LIN {X 0,Y 528.521,Z 608.402,A -85,B 0,C 180,E1 23622.926,E2 23622.926} C_VEL
LIN {X 0,Y 528.515,Z 608.398,A -85,B 0,C 180,E1 23619.468,E2 23619.468} C_VEL
LIN {X 0,Y 528.508,Z 608.399,A -85,B 0,C 180,E1 23616.041,E2 23616.041} C_VEL
LIN {X 0,Y 528.521,Z 608.403,A -85,B 0,C 180,E1 23612.627,E2 23612.627} C_VEL
LIN {X 0,Y 528.529,Z 608.395,A -85,B 0,C 180,E1 23609.214,E2 23609.214} C_VEL
LIN {X 0,Y 528.495,Z 608.401,A -85,B 0,C 180,E1 23605.77,E2 23605.77} C_VEL
LIN {X 0,Y 528.522,Z 608.404,A -85,B 0,C 180,E1 23602.317,E2 23602.317} C_VEL
LIN {X 0,Y 528.519,Z 608.398,A -85,B 0,C 180,E1 23598.875,E2 23598.875} C_VEL
LIN {X 0,Y 528.48,Z 608.403,A -85,B 0,C 180,E1 23595.472,E2 23595.472} C_VEL
LIN {X 0,Y 528.523,Z 608.403,A -85,B 0,C 180,E1 23592.122,E2 23592.122} C_VEL
LIN {X 0,Y 528.485,Z 608.404,A -85,B 0,C 180,E1 23588.815,E2 23588.815} C_VEL
LIN {X 0,Y 528.558,Z 608.653,A -85,B 0,C 180,E1 23586.299,E2 23586.299} C_VEL
LIN {X 0,Y 531.147,Z 620.669,A -85,B 0,C 180,E1 23584.859,E2 23584.859} C_VEL
LIN {X 0,Y 531.113,Z 646.994,A -85,B 0,C 180,E1 23581.942,E2 23581.942} C_VEL
LIN {X 0,Y 530.812,Z 675.191,A -85,B 0,C 180,E1 23578.705,E2 23578.705} C_VEL
LIN {X 0,Y 530.502,Z 697.757,A -85,B 0,C 180,E1 23576.089,E2 23576.089} C_VEL
LIN {X 0,Y 531.315,Z 704.19,A -85,B 0,C 180,E1 23575.96,E2 23575.96} C_VEL
LIN {X 0,Y 530.592,Z 836.819,A -85,B 0,C 180,E1 23574.081,E2 23574.081} C_VEL
LIN {X 0,Y 530.428,Z 853.085,A -85,B 0,C 180,E1 23573.642,E2 23573.642} C_VEL
LIN {X 0,Y 530.169,Z 868.62,A -85,B 0,C 180,E1 23573.013,E2 23573.013} C_VEL
LIN {X 0,Y 529.83,Z 883.45,A -85,B 0,C 180,E1 23572.191,E2 23572.191} C_VEL
LIN {X 0,Y 529.463,Z 897.184,A -85,B 0,C 180,E1 23571.201,E2 23571.201} C_VEL
LIN {X 0,Y 529.097,Z 909.864,A -85,B 0,C 180,E1 23570.043,E2 23570.043} C_VEL
LIN {X 0,Y 528.754,Z 921.003,A -85,B 0,C 180,E1 23568.768,E2 23568.768} C_VEL
LIN {X 0,Y 528.457,Z 931.118,A -85,B 0,C 180,E1 23567.322,E2 23567.322} C_VEL
LIN {X 0,Y 528.239,Z 939.83,A -85,B 0,C 180,E1 23565.726,E2 23565.726} C_VEL
LIN {X 0,Y 528.101,Z 946.573,A -85,B 0,C 180,E1 23564.114,E2 23564.114} C_VEL
LIN {X 0,Y 528.006,Z 952.107,A -85,B 0,C 180,E1 23562.272,E2 23562.272} C_VEL
LIN {X 0,Y 528.005,Z 952.163,A -85,B 0,C 180,E1 23562.25,E2 23562.25} C_VEL
LIN {X 0,Y 526.984,Z 954.183,A -85,B 0,C 180,E1 23561.442,E2 23561.442} C_VEL
LIN {X 0,Y 522.729,Z 957.032,A -85,B 0,C 180,E1 23560.019,E2 23560.019} C_VEL
LIN {X 0,Y 520.31,Z 958.175,A -85,B 0,C 180,E1 23558.953,E2 23558.953} C_VEL
LIN {X 0,Y 520.045,Z 958.343,A -85,B 0,C 180,E1 23558.525,E2 23558.525} C_VEL
LIN {X 0,Y 520.041,Z 957.958,A -85,B 0,C 180,E1 23556.667,E2 23556.667} C_VEL
LIN {X 0,Y 520.063,Z 955.8,A -85,B 0,C 180,E1 23554.856,E2 23554.856} C_VEL
LIN {X 0,Y 520.12,Z 951.746,A -85,B 0,C 180,E1 23553.02,E2 23553.02} C_VEL
LIN {X 0,Y 520.236,Z 945.996,A -85,B 0,C 180,E1 23551.283,E2 23551.283} C_VEL
LIN {X 0,Y 520.411,Z 938.536,A -85,B 0,C 180,E1 23549.617,E2 23549.617} C_VEL
LIN {X 0,Y 520.663,Z 929.608,A -85,B 0,C 180,E1 23548.082,E2 23548.082} C_VEL
LIN {X 0,Y 521.01,Z 918.657,A -85,B 0,C 180,E1 23546.596,E2 23546.596} C_VEL
LIN {X 0,Y 521.408,Z 906.398,A -85,B 0,C 180,E1 23545.282,E2 23545.282} C_VEL
LIN {X 0,Y 521.806,Z 893.101,A -85,B 0,C 180,E1 23544.149,E2 23544.149} C_VEL
LIN {X 0,Y 522.198,Z 878.496,A -85,B 0,C 180,E1 23543.179,E2 23543.179} C_VEL
LIN {X 0,Y 522.544,Z 863.741,A -85,B 0,C 180,E1 23542.434,E2 23542.434} C_VEL
LIN {X 0,Y 522.797,Z 847.6,A -85,B 0,C 180,E1 23541.853,E2 23541.853} C_VEL
LIN {X 0,Y 522.937,Z 831.072,A -85,B 0,C 180,E1 23541.478,E2 23541.478} C_VEL
LIN {X 0,Y 523.508,Z 702.169,A -85,B 0,C 180,E1 23539.641,E2 23539.641} C_VEL
LIN {X 0,Y 522.522,Z 696.556,A -85,B 0,C 180,E1 23539.485,E2 23539.485} C_VEL
LIN {X 0,Y 523.125,Z 666.461,A -85,B 0,C 180,E1 23535.915,E2 23535.915} C_VEL
LIN {X 0,Y 523.521,Z 639.644,A -85,B 0,C 180,E1 23532.766,E2 23532.766} C_VEL
LIN {X 0,Y 523.551,Z 621.942,A -85,B 0,C 180,E1 23530.696,E2 23530.696} C_VEL
LIN {X 0,Y 520.538,Z 609.538,A -85,B 0,C 180,E1 23529.053,E2 23529.053} C_VEL
LIN {X 0,Y 520.56,Z 609.378,A -85,B 0,C 180,E1 23525.998,E2 23525.998} C_VEL
LIN {X 0,Y 520.521,Z 609.389,A -85,B 0,C 180,E1 23522.668,E2 23522.668} C_VEL
LIN {X 0,Y 520.586,Z 609.388,A -85,B 0,C 180,E1 23519.311,E2 23519.311} C_VEL
LIN {X 0,Y 520.535,Z 609.391,A -85,B 0,C 180,E1 23515.979,E2 23515.979} C_VEL
LIN {X 0,Y 520.536,Z 609.392,A -85,B 0,C 180,E1 23512.473,E2 23512.473} C_VEL
LIN {X 0,Y 520.583,Z 609.379,A -85,B 0,C 180,E1 23509.174,E2 23509.174} C_VEL
LIN {X 0,Y 520.532,Z 609.381,A -85,B 0,C 180,E1 23505.829,E2 23505.829} C_VEL
LIN {X 0,Y 520.625,Z 609.66,A -85,B 0,C 180,E1 23502.669,E2 23502.669} C_VEL
LIN {X 0,Y 524.764,Z 625.278,A -85,B 0,C 180,E1 23500.318,E2 23500.318} C_VEL
LIN {X 0,Y 523.759,Z 651.946,A -85,B 0,C 180,E1 23496.908,E2 23496.908} C_VEL
LIN {X 0,Y 522.864,Z 678.978,A -85,B 0,C 180,E1 23493.509,E2 23493.509} C_VEL
LIN {X 0,Y 522.468,Z 693.224,A -85,B 0,C 180,E1 23491.755,E2 23491.755} C_VEL
LIN {X 0,Y 524.511,Z 704.529,A -85,B 0,C 180,E1 23491.475,E2 23491.475} C_VEL
LIN {X 0,Y 523.61,Z 835.562,A -85,B 0,C 180,E1 23489.587,E2 23489.587} C_VEL
LIN {X 0,Y 523.359,Z 852.526,A -85,B 0,C 180,E1 23489.121,E2 23489.121} C_VEL
LIN {X 0,Y 523.024,Z 867.254,A -85,B 0,C 180,E1 23488.521,E2 23488.521} C_VEL
LIN {X 0,Y 522.574,Z 882.116,A -85,B 0,C 180,E1 23487.698,E2 23487.698} C_VEL
LIN {X 0,Y 522.088,Z 896.006,A -85,B 0,C 180,E1 23486.707,E2 23486.707} C_VEL
LIN {X 0,Y 521.613,Z 908.793,A -85,B 0,C 180,E1 23485.548,E2 23485.548} C_VEL
LIN {X 0,Y 521.147,Z 920.994,A -85,B 0,C 180,E1 23484.164,E2 23484.164} C_VEL
LIN {X 0,Y 520.756,Z 931.108,A -85,B 0,C 180,E1 23482.72,E2 23482.72} C_VEL
LIN {X 0,Y 520.453,Z 940.34,A -85,B 0,C 180,E1 23481.048,E2 23481.048} C_VEL
LIN {X 0,Y 520.258,Z 947.386,A -85,B 0,C 180,E1 23479.368,E2 23479.368} C_VEL
LIN {X 0,Y 520.15,Z 952.932,A -85,B 0,C 180,E1 23477.557,E2 23477.557} C_VEL
LIN {X 0,Y 520.084,Z 956.511,A -85,B 0,C 180,E1 23475.755,E2 23475.755} C_VEL
LIN {X 0,Y 520.059,Z 958.338,A -85,B 0,C 180,E1 23473.928,E2 23473.928} C_VEL
LIN {X 0,Y 520.062,Z 958.416,A -85,B 0,C 180,E1 23472.085,E2 23472.085} C_VEL
LIN {X 0,Y 520.09,Z 956.657,A -85,B 0,C 180,E1 23470.224,E2 23470.224} C_VEL
LIN {X 0,Y 520.157,Z 953.294,A -85,B 0,C 180,E1 23468.461,E2 23468.461} C_VEL
LIN {X 0,Y 520.269,Z 947.993,A -85,B 0,C 180,E1 23466.679,E2 23466.679} C_VEL
LIN {X 0,Y 520.461,Z 941.165,A -85,B 0,C 180,E1 23464.999,E2 23464.999} C_VEL
LIN {X 0,Y 520.742,Z 932.761,A -85,B 0,C 180,E1 23463.425,E2 23463.425} C_VEL
LIN {X 0,Y 521.128,Z 922.872,A -85,B 0,C 180,E1 23461.955,E2 23461.955} C_VEL
LIN {X 0,Y 521.583,Z 911.544,A -85,B 0,C 180,E1 23460.611,E2 23460.611} C_VEL
LIN {X 0,Y 522.08,Z 898.49,A -85,B 0,C 180,E1 23459.374,E2 23459.374} C_VEL
LIN {X 0,Y 522.567,Z 885.129,A -85,B 0,C 180,E1 23458.37,E2 23458.37} C_VEL
LIN {X 0,Y 523.027,Z 870.3,A -85,B 0,C 180,E1 23457.508,E2 23457.508} C_VEL
LIN {X 0,Y 523.414,Z 855.24,A -85,B 0,C 180,E1 23456.852,E2 23456.852} C_VEL
LIN {X 0,Y 523.674,Z 839.22,A -85,B 0,C 180,E1 23456.375,E2 23456.375} C_VEL
LIN {X 0,Y 523.861,Z 816.787,A -85,B 0,C 180,E1 23455.998,E2 23455.998} C_VEL
LIN {X 0,Y 524.467,Z 702.284,A -85,B 0,C 180,E1 23454.351,E2 23454.351} C_VEL
LIN {X 0,Y 522.558,Z 693.202,A -85,B 0,C 180,E1 23454.094,E2 23454.094} C_VEL
LIN {X 0,Y 523.474,Z 665.562,A -85,B 0,C 180,E1 23450.644,E2 23450.644} C_VEL
LIN {X 0,Y 524.54,Z 637.445,A -85,B 0,C 180,E1 23447.052,E2 23447.052} C_VEL
LIN {X 0,Y 524.869,Z 625.09,A -85,B 0,C 180,E1 23445.436,E2 23445.436} C_VEL
LIN {X 0,Y 520.594,Z 609.506,A -85,B 0,C 180,E1 23442.986,E2 23442.986} C_VEL
LIN {X 0,Y 520.574,Z 609.387,A -85,B 0,C 180,E1 23439.456,E2 23439.456} C_VEL
LIN {X 0,Y 520.573,Z 609.389,A -85,B 0,C 180,E1 23435.997,E2 23435.997} C_VEL
LIN {X 0,Y 520.583,Z 609.393,A -85,B 0,C 180,E1 23432.524,E2 23432.524} C_VEL
LIN {X 0,Y 520.58,Z 609.385,A -85,B 0,C 180,E1 23429.074,E2 23429.074} C_VEL
LIN {X 0,Y 520.57,Z 609.385,A -85,B 0,C 180,E1 23425.605,E2 23425.605} C_VEL
LIN {X 0,Y 520.586,Z 609.386,A -85,B 0,C 180,E1 23422.114,E2 23422.114} C_VEL
LIN {X 0,Y 520.579,Z 609.382,A -85,B 0,C 180,E1 23418.593,E2 23418.593} C_VEL
LIN {X 0,Y 520.566,Z 609.383,A -85,B 0,C 180,E1 23415.143,E2 23415.143} C_VEL
LIN {X 0,Y 520.581,Z 609.391,A -85,B 0,C 180,E1 23411.635,E2 23411.635} C_VEL
LIN {X 0,Y 520.581,Z 609.385,A -85,B 0,C 180,E1 23408.171,E2 23408.171} C_VEL
LIN {X 0,Y 520.565,Z 609.386,A -85,B 0,C 180,E1 23404.738,E2 23404.738} C_VEL
LIN {X 0,Y 520.582,Z 609.385,A -85,B 0,C 180,E1 23401.321,E2 23401.321} C_VEL
LIN {X 0,Y 520.583,Z 609.384,A -85,B 0,C 180,E1 23397.799,E2 23397.799} C_VEL
LIN {X 0,Y 520.563,Z 609.387,A -85,B 0,C 180,E1 23394.379,E2 23394.379} C_VEL
LIN {X 0,Y 520.582,Z 609.382,A -85,B 0,C 180,E1 23390.939,E2 23390.939} C_VEL
LIN {X 0,Y 520.584,Z 609.383,A -85,B 0,C 180,E1 23387.465,E2 23387.465} C_VEL
LIN {X 0,Y 520.562,Z 609.391,A -85,B 0,C 180,E1 23384.058,E2 23384.058} C_VEL
LIN {X 0,Y 520.581,Z 609.38,A -85,B 0,C 180,E1 23380.71,E2 23380.71} C_VEL
LIN {X 0,Y 520.566,Z 609.381,A -85,B 0,C 180,E1 23377.29,E2 23377.29} C_VEL
LIN {X 0,Y 520.567,Z 609.387,A -85,B 0,C 180,E1 23373.762,E2 23373.762} C_VEL
LIN {X 0,Y 520.582,Z 609.389,A -85,B 0,C 180,E1 23370.296,E2 23370.296} C_VEL
LIN {X 0,Y 520.564,Z 609.387,A -85,B 0,C 180,E1 23366.87,E2 23366.87} C_VEL
LIN {X 0,Y 520.565,Z 609.391,A -85,B 0,C 180,E1 23363.32,E2 23363.32} C_VEL
LIN {X 0,Y 520.584,Z 609.389,A -85,B 0,C 180,E1 23359.953,E2 23359.953} C_VEL
LIN {X 0,Y 520.557,Z 609.385,A -85,B 0,C 180,E1 23356.555,E2 23356.555} C_VEL
LIN {X 0,Y 520.578,Z 609.392,A -85,B 0,C 180,E1 23353.126,E2 23353.126} C_VEL
LIN {X 0,Y 520.587,Z 609.386,A -85,B 0,C 180,E1 23349.63,E2 23349.63} C_VEL
LIN {X 0,Y 520.553,Z 609.393,A -85,B 0,C 180,E1 23346.223,E2 23346.223} C_VEL
LIN {X 0,Y 520.617,Z 609.623,A -85,B 0,C 180,E1 23345.548,E2 23345.548} C_VEL
LIN {X 0,Y 528.314,Z 631.638,A -85,B 0,C 180,E1 23343.125,E2 23343.125} C_VEL
LIN {X 0,Y 526.952,Z 675.578,A -85,B 0,C 180,E1 23339.685,E2 23339.685} C_VEL
LIN {X 0,Y 525.974,Z 709.847,A -85,B 0,C 180,E1 23337.075,E2 23337.075} C_VEL
LIN {X 0,Y 527.931,Z 723.514,A -85,B 0,C 180,E1 23336.758,E2 23336.758} C_VEL
LIN {X 0,Y 526.233,Z 927.53,A -85,B 0,C 180,E1 23333.802,E2 23333.802} C_VEL
LIN {X 0,Y 525.783,Z 946.957,A -85,B 0,C 180,E1 23333.314,E2 23333.314} C_VEL
LIN {X 0,Y 525.229,Z 964.796,A -85,B 0,C 180,E1 23332.674,E2 23332.674} C_VEL
LIN {X 0,Y 524.559,Z 982.787,A -85,B 0,C 180,E1 23331.82,E2 23331.82} C_VEL
LIN {X 0,Y 523.785,Z 1000.784,A -85,B 0,C 180,E1 23330.732,E2 23330.732} C_VEL
LIN {X 0,Y 523.028,Z 1017.39,A -85,B 0,C 180,E1 23329.492,E2 23329.492} C_VEL
LIN {X 0,Y 522.315,Z 1032.415,A -85,B 0,C 180,E1 23328.137,E2 23328.137} C_VEL
LIN {X 0,Y 521.648,Z 1046.702,A -85,B 0,C 180,E1 23326.592,E2 23326.592} C_VEL
LIN {X 0,Y 521.078,Z 1059.756,A -85,B 0,C 180,E1 23324.899,E2 23324.899} C_VEL
LIN {X 0,Y 520.633,Z 1071.3,A -85,B 0,C 180,E1 23323.098,E2 23323.098} C_VEL
LIN {X 0,Y 520.313,Z 1081.338,A -85,B 0,C 180,E1 23321.191,E2 23321.191} C_VEL
LIN {X 0,Y 520.102,Z 1089.433,A -85,B 0,C 180,E1 23319.293,E2 23319.293} C_VEL
LIN {X 0,Y 519.989,Z 1096.129,A -85,B 0,C 180,E1 23317.291,E2 23317.291} C_VEL
LIN {X 0,Y 519.926,Z 1101.295,A -85,B 0,C 180,E1 23315.185,E2 23315.185} C_VEL
LIN {X 0,Y 519.912,Z 1104.658,A -85,B 0,C 180,E1 23313.086,E2 23313.086} C_VEL
LIN {X 0,Y 519.908,Z 1106.304,A -85,B 0,C 180,E1 23310.991,E2 23310.991} C_VEL
LIN {X 0,Y 519.906,Z 1106.265,A -85,B 0,C 180,E1 23308.898,E2 23308.898} C_VEL
LIN {X 0,Y 519.914,Z 1104.539,A -85,B 0,C 180,E1 23306.803,E2 23306.803} C_VEL
LIN {X 0,Y 519.927,Z 1101.085,A -85,B 0,C 180,E1 23304.703,E2 23304.703} C_VEL
LIN {X 0,Y 519.992,Z 1095.818,A -85,B 0,C 180,E1 23302.598,E2 23302.598} C_VEL
LIN {X 0,Y 520.129,Z 1088.591,A -85,B 0,C 180,E1 23300.484,E2 23300.484} C_VEL
LIN {X 0,Y 520.358,Z 1079.733,A -85,B 0,C 180,E1 23298.472,E2 23298.472} C_VEL
LIN {X 0,Y 520.706,Z 1069.307,A -85,B 0,C 180,E1 23296.565,E2 23296.565} C_VEL
LIN {X 0,Y 521.168,Z 1057.586,A -85,B 0,C 180,E1 23294.797,E2 23294.797} C_VEL
LIN {X 0,Y 521.745,Z 1044.4,A -85,B 0,C 180,E1 23293.141,E2 23293.141} C_VEL
LIN {X 0,Y 522.396,Z 1030.569,A -85,B 0,C 180,E1 23291.684,E2 23291.684} C_VEL
LIN {X 0,Y 523.121,Z 1015.357,A -85,B 0,C 180,E1 23290.342,E2 23290.342} C_VEL
LIN {X 0,Y 523.869,Z 998.977,A -85,B 0,C 180,E1 23289.148,E2 23289.148} C_VEL
LIN {X 0,Y 524.599,Z 981.79,A -85,B 0,C 180,E1 23288.129,E2 23288.129} C_VEL
LIN {X 0,Y 525.255,Z 963.935,A -85,B 0,C 180,E1 23287.291,E2 23287.291} C_VEL
LIN {X 0,Y 525.829,Z 944.794,A -85,B 0,C 180,E1 23286.621,E2 23286.621} C_VEL
LIN {X 0,Y 526.261,Z 925.545,A -85,B 0,C 180,E1 23286.162,E2 23286.162} C_VEL
LIN {X 0,Y 527.774,Z 721.067,A -85,B 0,C 180,E1 23283.197,E2 23283.197} C_VEL
LIN {X 0,Y 525.911,Z 709.157,A -85,B 0,C 180,E1 23282.898,E2 23282.898} C_VEL
LIN {X 0,Y 527.325,Z 664.166,A -85,B 0,C 180,E1 23279.409,E2 23279.409} C_VEL
LIN {X 0,Y 528.418,Z 631.682,A -85,B 0,C 180,E1 23276.849,E2 23276.849} C_VEL
LIN {X 0,Y 520.631,Z 609.705,A -85,B 0,C 180,E1 23274.452,E2 23274.452} C_VEL
LIN {X 0,Y 520.581,Z 609.389,A -85,B 0,C 180,E1 23273.184,E2 23273.184} C_VEL
LIN {X 0,Y 520.563,Z 609.39,A -85,B 0,C 180,E1 23269.687,E2 23269.687} C_VEL
LIN {X 0,Y 520.582,Z 609.384,A -85,B 0,C 180,E1 23266.234,E2 23266.234} C_VEL
LIN {X 0,Y 520.58,Z 609.391,A -85,B 0,C 180,E1 23262.687,E2 23262.687} C_VEL
LIN {X 0,Y 520.573,Z 609.389,A -85,B 0,C 180,E1 23259.281,E2 23259.281} C_VEL
LIN {X 0,Y 520.574,Z 609.386,A -85,B 0,C 180,E1 23255.852,E2 23255.852} C_VEL
LIN {X 0,Y 520.569,Z 609.391,A -85,B 0,C 180,E1 23252.273,E2 23252.273} C_VEL
LIN {X 0,Y 520.583,Z 609.389,A -85,B 0,C 180,E1 23248.821,E2 23248.821} C_VEL
LIN {X 0,Y 520.571,Z 609.387,A -85,B 0,C 180,E1 23245.361,E2 23245.361} C_VEL
LIN {X 0,Y 520.556,Z 609.392,A -85,B 0,C 180,E1 23241.877,E2 23241.877} C_VEL
LIN {X 0,Y 520.588,Z 609.39,A -85,B 0,C 180,E1 23238.476,E2 23238.476} C_VEL
LIN {X 0,Y 520.547,Z 609.391,A -85,B 0,C 180,E1 23235.143,E2 23235.143} C_VEL
LIN {X 0,Y 520.546,Z 609.395,A -85,B 0,C 180,E1 23231.59,E2 23231.59} C_VEL
LIN {X 0,Y 520.59,Z 609.391,A -85,B 0,C 180,E1 23228.171,E2 23228.171} C_VEL
LIN {X 0,Y 520.576,Z 609.575,A -85,B 0,C 180,E1 23226.617,E2 23226.617} C_VEL
LIN {X 0,Y 523.556,Z 623.071,A -85,B 0,C 180,E1 23224.985,E2 23224.985} C_VEL
LIN {X 0,Y 523.519,Z 650.254,A -85,B 0,C 180,E1 23221.97,E2 23221.97} C_VEL
LIN {X 0,Y 523.179,Z 679.795,A -85,B 0,C 180,E1 23218.576,E2 23218.576} C_VEL
LIN {X 0,Y 522.952,Z 699.166,A -85,B 0,C 180,E1 23216.344,E2 23216.344} C_VEL
LIN {X 0,Y 523.715,Z 705.163,A -85,B 0,C 180,E1 23216.221,E2 23216.221} C_VEL
LIN {X 0,Y 522.897,Z 838.188,A -85,B 0,C 180,E1 23214.297,E2 23214.297} C_VEL
LIN {X 0,Y 522.743,Z 854.027,A -85,B 0,C 180,E1 23213.865,E2 23213.865} C_VEL
LIN {X 0,Y 522.484,Z 869.358,A -85,B 0,C 180,E1 23213.241,E2 23213.241} C_VEL
LIN {X 0,Y 522.159,Z 883.503,A -85,B 0,C 180,E1 23212.463,E2 23212.463} C_VEL
LIN {X 0,Y 521.753,Z 897.813,A -85,B 0,C 180,E1 23211.433,E2 23211.433} C_VEL
LIN {X 0,Y 521.369,Z 910.395,A -85,B 0,C 180,E1 23210.284,E2 23210.284} C_VEL
LIN {X 0,Y 520.977,Z 922.127,A -85,B 0,C 180,E1 23208.935,E2 23208.935} C_VEL
LIN {X 0,Y 520.646,Z 932.272,A -85,B 0,C 180,E1 23207.466,E2 23207.466} C_VEL
LIN {X 0,Y 520.402,Z 940.878,A -85,B 0,C 180,E1 23205.877,E2 23205.877} C_VEL
LIN {X 0,Y 520.243,Z 947.547,A -85,B 0,C 180,E1 23204.277,E2 23204.277} C_VEL
LIN {X 0,Y 520.123,Z 953.086,A -85,B 0,C 180,E1 23202.433,E2 23202.433} C_VEL
LIN {X 0,Y 520.066,Z 956.47,A -85,B 0,C 180,E1 23200.69,E2 23200.69} C_VEL
LIN {X 0,Y 520.042,Z 958.242,A -85,B 0,C 180,E1 23198.81,E2 23198.81} C_VEL
LIN {X 0,Y 520.045,Z 958.343,A -85,B 0,C 180,E1 23198.525,E2 23198.525} C_VEL
LIN {X 0,Y 519.064,Z 958.538,A -85,B 0,C 180,E1 23197.676,E2 23197.676} C_VEL
LIN {X 0,Y 514.653,Z 958.354,A -85,B 0,C 180,E1 23196.137,E2 23196.137} C_VEL
LIN {X 0,Y 512.417,Z 957.426,A -85,B 0,C 180,E1 23195.112,E2 23195.112} C_VEL
LIN {X 0,Y 512.16,Z 956.752,A -85,B 0,C 180,E1 23194.683,E2 23194.683} C_VEL
LIN {X 0,Y 512.236,Z 952.557,A -85,B 0,C 180,E1 23192.822,E2 23192.822} C_VEL
LIN {X 0,Y 512.369,Z 946.613,A -85,B 0,C 180,E1 23191.055,E2 23191.055} C_VEL
LIN {X 0,Y 512.573,Z 939.119,A -85,B 0,C 180,E1 23189.394,E2 23189.394} C_VEL
LIN {X 0,Y 512.867,Z 929.708,A -85,B 0,C 180,E1 23187.791,E2 23187.791} C_VEL
LIN {X 0,Y 513.246,Z 918.892,A -85,B 0,C 180,E1 23186.333,E2 23186.333} C_VEL
LIN {X 0,Y 513.67,Z 906.73,A -85,B 0,C 180,E1 23185.033,E2 23185.033} C_VEL
LIN {X 0,Y 514.072,Z 894.233,A -85,B 0,C 180,E1 23183.959,E2 23183.959} C_VEL
LIN {X 0,Y 514.47,Z 880.225,A -85,B 0,C 180,E1 23183.013,E2 23183.013} C_VEL
LIN {X 0,Y 514.849,Z 864.996,A -85,B 0,C 180,E1 23182.225,E2 23182.225} C_VEL
LIN {X 0,Y 515.107,Z 848.894,A -85,B 0,C 180,E1 23181.635,E2 23181.635} C_VEL
LIN {X 0,Y 515.252,Z 832.388,A -85,B 0,C 180,E1 23181.25,E2 23181.25} C_VEL
LIN {X 0,Y 515.9,Z 703.02,A -85,B 0,C 180,E1 23179.37,E2 23179.37} C_VEL
LIN {X 0,Y 514.903,Z 697.689,A -85,B 0,C 180,E1 23179.229,E2 23179.229} C_VEL
LIN {X 0,Y 515.501,Z 667.96,A -85,B 0,C 180,E1 23175.702,E2 23175.702} C_VEL
LIN {X 0,Y 515.964,Z 638.618,A -85,B 0,C 180,E1 23172.246,E2 23172.246} C_VEL
LIN {X 0,Y 515.968,Z 624.273,A -85,B 0,C 180,E1 23170.568,E2 23170.568} C_VEL
LIN {X 0,Y 512.598,Z 610.534,A -85,B 0,C 180,E1 23168.738,E2 23168.738} C_VEL
LIN {X 0,Y 512.635,Z 610.374,A -85,B 0,C 180,E1 23165.537,E2 23165.537} C_VEL
LIN {X 0,Y 512.595,Z 610.38,A -85,B 0,C 180,E1 23162.161,E2 23162.161} C_VEL
LIN {X 0,Y 512.591,Z 610.379,A -85,B 0,C 180,E1 23158.676,E2 23158.676} C_VEL
LIN {X 0,Y 512.641,Z 610.363,A -85,B 0,C 180,E1 23155.41,E2 23155.41} C_VEL
LIN {X 0,Y 512.591,Z 610.382,A -85,B 0,C 180,E1 23152.098,E2 23152.098} C_VEL
LIN {X 0,Y 512.626,Z 610.376,A -85,B 0,C 180,E1 23148.656,E2 23148.656} C_VEL
LIN {X 0,Y 512.626,Z 610.369,A -85,B 0,C 180,E1 23145.267,E2 23145.267} C_VEL
LIN {X 0,Y 512.676,Z 610.651,A -85,B 0,C 180,E1 23143.076,E2 23143.076} C_VEL
LIN {X 0,Y 517.224,Z 627.697,A -85,B 0,C 180,E1 23140.47,E2 23140.47} C_VEL
LIN {X 0,Y 516.176,Z 653.615,A -85,B 0,C 180,E1 23137.122,E2 23137.122} C_VEL
LIN {X 0,Y 515.201,Z 680.751,A -85,B 0,C 180,E1 23133.672,E2 23133.672} C_VEL
LIN {X 0,Y 514.831,Z 693.315,A -85,B 0,C 180,E1 23132.115,E2 23132.115} C_VEL
LIN {X 0,Y 517.116,Z 705.629,A -85,B 0,C 180,E1 23131.799,E2 23131.799} C_VEL
LIN {X 0,Y 516.122,Z 836.216,A -85,B 0,C 180,E1 23129.889,E2 23129.889} C_VEL
LIN {X 0,Y 515.853,Z 853.205,A -85,B 0,C 180,E1 23129.417,E2 23129.417} C_VEL
LIN {X 0,Y 515.472,Z 868.6,A -85,B 0,C 180,E1 23128.778,E2 23128.778} C_VEL
LIN {X 0,Y 514.985,Z 883.365,A -85,B 0,C 180,E1 23127.942,E2 23127.942} C_VEL
LIN {X 0,Y 514.456,Z 897.202,A -85,B 0,C 180,E1 23126.937,E2 23126.937} C_VEL
LIN {X 0,Y 513.93,Z 909.944,A -85,B 0,C 180,E1 23125.761,E2 23125.761} C_VEL
LIN {X 0,Y 513.414,Z 922.076,A -85,B 0,C 180,E1 23124.363,E2 23124.363} C_VEL
LIN {X 0,Y 512.99,Z 931.894,A -85,B 0,C 180,E1 23122.947,E2 23122.947} C_VEL
LIN {X 0,Y 512.634,Z 941.187,A -85,B 0,C 180,E1 23121.25,E2 23121.25} C_VEL
LIN {X 0,Y 512.4,Z 948.32,A -85,B 0,C 180,E1 23119.545,E2 23119.545} C_VEL
LIN {X 0,Y 512.266,Z 953.893,A -85,B 0,C 180,E1 23117.717,E2 23117.717} C_VEL
LIN {X 0,Y 512.187,Z 957.444,A -85,B 0,C 180,E1 23115.982,E2 23115.982} C_VEL
LIN {X 0,Y 512.15,Z 959.408,A -85,B 0,C 180,E1 23114.138,E2 23114.138} C_VEL
LIN {X 0,Y 512.15,Z 959.693,A -85,B 0,C 180,E1 23112.269,E2 23112.269} C_VEL
LIN {X 0,Y 512.183,Z 958.134,A -85,B 0,C 180,E1 23110.381,E2 23110.381} C_VEL
LIN {X 0,Y 512.267,Z 954.706,A -85,B 0,C 180,E1 23108.473,E2 23108.473} C_VEL
LIN {X 0,Y 512.394,Z 949.948,A -85,B 0,C 180,E1 23106.786,E2 23106.786} C_VEL
LIN {X 0,Y 512.62,Z 942.814,A -85,B 0,C 180,E1 23104.96,E2 23104.96} C_VEL
LIN {X 0,Y 512.944,Z 934.596,A -85,B 0,C 180,E1 23103.364,E2 23103.364} C_VEL
LIN {X 0,Y 513.406,Z 924.011,A -85,B 0,C 180,E1 23101.755,E2 23101.755} C_VEL
LIN {X 0,Y 513.916,Z 912.644,A -85,B 0,C 180,E1 23100.385,E2 23100.385} C_VEL
LIN {X 0,Y 514.467,Z 899.608,A -85,B 0,C 180,E1 23099.131,E2 23099.131} C_VEL
LIN {X 0,Y 514.997,Z 886.471,A -85,B 0,C 180,E1 23098.124,E2 23098.124} C_VEL
LIN {X 0,Y 515.503,Z 871.529,A -85,B 0,C 180,E1 23097.239,E2 23097.239} C_VEL
LIN {X 0,Y 515.941,Z 855.774,A -85,B 0,C 180,E1 23096.541,E2 23096.541} C_VEL
LIN {X 0,Y 516.213,Z 839.686,A -85,B 0,C 180,E1 23096.061,E2 23096.061} C_VEL
LIN {X 0,Y 516.413,Z 816.95,A -85,B 0,C 180,E1 23095.676,E2 23095.676} C_VEL
LIN {X 0,Y 517.106,Z 703.505,A -85,B 0,C 180,E1 23094.018,E2 23094.018} C_VEL
LIN {X 0,Y 514.98,Z 693.607,A -85,B 0,C 180,E1 23093.743,E2 23093.743} C_VEL
LIN {X 0,Y 515.872,Z 668.015,A -85,B 0,C 180,E1 23090.526,E2 23090.526} C_VEL
LIN {X 0,Y 517.05,Z 639.818,A -85,B 0,C 180,E1 23086.875,E2 23086.875} C_VEL
LIN {X 0,Y 517.462,Z 627.908,A -85,B 0,C 180,E1 23085.305,E2 23085.305} C_VEL
LIN {X 0,Y 512.672,Z 610.626,A -85,B 0,C 180,E1 23082.553,E2 23082.553} C_VEL
LIN {X 0,Y 512.632,Z 610.379,A -85,B 0,C 180,E1 23079.194,E2 23079.194} C_VEL
LIN {X 0,Y 512.643,Z 610.375,A -85,B 0,C 180,E1 23075.674,E2 23075.674} C_VEL
LIN {X 0,Y 512.637,Z 610.377,A -85,B 0,C 180,E1 23072.169,E2 23072.169} C_VEL
LIN {X 0,Y 512.636,Z 610.376,A -85,B 0,C 180,E1 23068.673,E2 23068.673} C_VEL
LIN {X 0,Y 512.643,Z 610.37,A -85,B 0,C 180,E1 23065.163,E2 23065.163} C_VEL
LIN {X 0,Y 512.634,Z 610.378,A -85,B 0,C 180,E1 23061.632,E2 23061.632} C_VEL
LIN {X 0,Y 512.637,Z 610.373,A -85,B 0,C 180,E1 23058.184,E2 23058.184} C_VEL
LIN {X 0,Y 512.649,Z 610.367,A -85,B 0,C 180,E1 23054.674,E2 23054.674} C_VEL
LIN {X 0,Y 512.628,Z 610.373,A -85,B 0,C 180,E1 23051.134,E2 23051.134} C_VEL
LIN {X 0,Y 512.643,Z 610.38,A -85,B 0,C 180,E1 23047.622,E2 23047.622} C_VEL
LIN {X 0,Y 512.642,Z 610.372,A -85,B 0,C 180,E1 23044.027,E2 23044.027} C_VEL
LIN {X 0,Y 512.625,Z 610.37,A -85,B 0,C 180,E1 23040.559,E2 23040.559} C_VEL
LIN {X 0,Y 512.643,Z 610.376,A -85,B 0,C 180,E1 23037.093,E2 23037.093} C_VEL
LIN {X 0,Y 512.644,Z 610.373,A -85,B 0,C 180,E1 23033.505,E2 23033.505} C_VEL
LIN {X 0,Y 512.624,Z 610.373,A -85,B 0,C 180,E1 23030.059,E2 23030.059} C_VEL
LIN {X 0,Y 512.644,Z 610.372,A -85,B 0,C 180,E1 23026.58,E2 23026.58} C_VEL
LIN {X 0,Y 512.645,Z 610.375,A -85,B 0,C 180,E1 23023.106,E2 23023.106} C_VEL
LIN {X 0,Y 512.623,Z 610.378,A -85,B 0,C 180,E1 23019.685,E2 23019.685} C_VEL
LIN {X 0,Y 512.643,Z 610.373,A -85,B 0,C 180,E1 23016.188,E2 23016.188} C_VEL
LIN {X 0,Y 512.645,Z 610.369,A -85,B 0,C 180,E1 23012.72,E2 23012.72} C_VEL
LIN {X 0,Y 512.619,Z 610.372,A -85,B 0,C 180,E1 23009.268,E2 23009.268} C_VEL
LIN {X 0,Y 512.646,Z 610.376,A -85,B 0,C 180,E1 23005.788,E2 23005.788} C_VEL
LIN {X 0,Y 512.647,Z 610.373,A -85,B 0,C 180,E1 23002.235,E2 23002.235} C_VEL
LIN {X 0,Y 512.617,Z 610.378,A -85,B 0,C 180,E1 22998.841,E2 22998.841} C_VEL
LIN {X 0,Y 512.645,Z 610.379,A -85,B 0,C 180,E1 22995.389,E2 22995.389} C_VEL
LIN {X 0,Y 512.644,Z 610.375,A -85,B 0,C 180,E1 22991.837,E2 22991.837} C_VEL
LIN {X 0,Y 512.614,Z 610.379,A -85,B 0,C 180,E1 22988.362,E2 22988.362} C_VEL
LIN {X 0,Y 512.657,Z 610.649,A -85,B 0,C 180,E1 22986.029,E2 22986.029} C_VEL
LIN {X 0,Y 519.677,Z 630.467,A -85,B 0,C 180,E1 22983.781,E2 22983.781} C_VEL
LIN {X 0,Y 521.03,Z 634.412,A -85,B 0,C 180,E1 22983.359,E2 22983.359} C_VEL
LIN {X 0,Y 519.493,Z 677.903,A -85,B 0,C 180,E1 22979.9,E2 22979.9} C_VEL
LIN {X 0,Y 518.492,Z 709.662,A -85,B 0,C 180,E1 22977.451,E2 22977.451} C_VEL
LIN {X 0,Y 520.724,Z 724.661,A -85,B 0,C 180,E1 22977.125,E2 22977.125} C_VEL
LIN {X 0,Y 518.917,Z 927.366,A -85,B 0,C 180,E1 22974.162,E2 22974.162} C_VEL
LIN {X 0,Y 518.422,Z 946.848,A -85,B 0,C 180,E1 22973.669,E2 22973.669} C_VEL
LIN {X 0,Y 517.796,Z 965.228,A -85,B 0,C 180,E1 22972.998,E2 22972.998} C_VEL
LIN {X 0,Y 517.076,Z 982.901,A -85,B 0,C 180,E1 22972.145,E2 22972.145} C_VEL
LIN {X 0,Y 516.233,Z 1000.7,A -85,B 0,C 180,E1 22971.056,E2 22971.056} C_VEL
LIN {X 0,Y 515.39,Z 1017.346,A -85,B 0,C 180,E1 22969.797,E2 22969.797} C_VEL
LIN {X 0,Y 514.59,Z 1032.543,A -85,B 0,C 180,E1 22968.405,E2 22968.405} C_VEL
LIN {X 0,Y 513.861,Z 1046.684,A -85,B 0,C 180,E1 22966.853,E2 22966.853} C_VEL
LIN {X 0,Y 513.225,Z 1059.757,A -85,B 0,C 180,E1 22965.133,E2 22965.133} C_VEL
LIN {X 0,Y 512.729,Z 1071.301,A -85,B 0,C 180,E1 22963.303,E2 22963.303} C_VEL
LIN {X 0,Y 512.364,Z 1081.339,A -85,B 0,C 180,E1 22961.367,E2 22961.367} C_VEL
LIN {X 0,Y 512.131,Z 1089.434,A -85,B 0,C 180,E1 22959.439,E2 22959.439} C_VEL
LIN {X 0,Y 511.997,Z 1096.129,A -85,B 0,C 180,E1 22957.405,E2 22957.405} C_VEL
LIN {X 0,Y 511.928,Z 1101.295,A -85,B 0,C 180,E1 22955.267,E2 22955.267} C_VEL
LIN {X 0,Y 511.913,Z 1104.657,A -85,B 0,C 180,E1 22953.135,E2 22953.135} C_VEL
LIN {X 0,Y 511.908,Z 1106.303,A -85,B 0,C 180,E1 22951.007,E2 22951.007} C_VEL
LIN {X 0,Y 511.906,Z 1106.265,A -85,B 0,C 180,E1 22948.881,E2 22948.881} C_VEL
LIN {X 0,Y 511.914,Z 1104.539,A -85,B 0,C 180,E1 22946.753,E2 22946.753} C_VEL
LIN {X 0,Y 511.931,Z 1101.085,A -85,B 0,C 180,E1 22944.62,E2 22944.62} C_VEL
LIN {X 0,Y 512.001,Z 1095.817,A -85,B 0,C 180,E1 22942.482,E2 22942.482} C_VEL
LIN {X 0,Y 512.159,Z 1088.59,A -85,B 0,C 180,E1 22940.334,E2 22940.334} C_VEL
LIN {X 0,Y 512.416,Z 1079.732,A -85,B 0,C 180,E1 22938.291,E2 22938.291} C_VEL
LIN {X 0,Y 512.806,Z 1069.306,A -85,B 0,C 180,E1 22936.354,E2 22936.354} C_VEL
LIN {X 0,Y 513.303,Z 1058.061,A -85,B 0,C 180,E1 22934.624,E2 22934.624} C_VEL
LIN {X 0,Y 513.952,Z 1044.739,A -85,B 0,C 180,E1 22932.916,E2 22932.916} C_VEL
LIN {X 0,Y 514.707,Z 1030.198,A -85,B 0,C 180,E1 22931.364,E2 22931.364} C_VEL
LIN {X 0,Y 515.515,Z 1014.819,A -85,B 0,C 180,E1 22929.996,E2 22929.996} C_VEL
LIN {X 0,Y 516.356,Z 998.084,A -85,B 0,C 180,E1 22928.77,E2 22928.77} C_VEL
LIN {X 0,Y 517.175,Z 980.554,A -85,B 0,C 180,E1 22927.732,E2 22927.732} C_VEL
LIN {X 0,Y 517.892,Z 962.601,A -85,B 0,C 180,E1 22926.896,E2 22926.896} C_VEL
LIN {X 0,Y 518.486,Z 944.051,A -85,B 0,C 180,E1 22926.248,E2 22926.248} C_VEL
LIN {X 0,Y 518.95,Z 924.903,A -85,B 0,C 180,E1 22925.793,E2 22925.793} C_VEL
LIN {X 0,Y 520.581,Z 722.325,A -85,B 0,C 180,E1 22922.834,E2 22922.834} C_VEL
LIN {X 0,Y 518.46,Z 708.947,A -85,B 0,C 180,E1 22922.513,E2 22922.513} C_VEL
LIN {X 0,Y 519.928,Z 664.783,A -85,B 0,C 180,E1 22919.058,E2 22919.058} C_VEL
LIN {X 0,Y 520.989,Z 634.108,A -85,B 0,C 180,E1 22916.598,E2 22916.598} C_VEL
LIN {X 0,Y 512.66,Z 610.644,A -85,B 0,C 180,E1 22913.951,E2 22913.951} C_VEL
LIN {X 0,Y 512.642,Z 610.381,A -85,B 0,C 180,E1 22910.742,E2 22910.742} C_VEL
LIN {X 0,Y 512.63,Z 610.379,A -85,B 0,C 180,E1 22907.334,E2 22907.334} C_VEL
LIN {X 0,Y 512.641,Z 610.372,A -85,B 0,C 180,E1 22903.809,E2 22903.809} C_VEL
LIN {X 0,Y 512.634,Z 610.378,A -85,B 0,C 180,E1 22900.304,E2 22900.304} C_VEL
LIN {X 0,Y 512.645,Z 610.381,A -85,B 0,C 180,E1 22896.782,E2 22896.782} C_VEL
LIN {X 0,Y 512.641,Z 610.376,A -85,B 0,C 180,E1 22893.203,E2 22893.203} C_VEL
LIN {X 0,Y 512.625,Z 610.376,A -85,B 0,C 180,E1 22889.777,E2 22889.777} C_VEL
LIN {X 0,Y 512.636,Z 610.381,A -85,B 0,C 180,E1 22886.279,E2 22886.279} C_VEL
LIN {X 0,Y 512.648,Z 610.376,A -85,B 0,C 180,E1 22882.838,E2 22882.838} C_VEL
LIN {X 0,Y 512.61,Z 610.379,A -85,B 0,C 180,E1 22879.484,E2 22879.484} C_VEL
LIN {X 0,Y 512.627,Z 610.383,A -85,B 0,C 180,E1 22875.963,E2 22875.963} C_VEL
LIN {X 0,Y 512.648,Z 610.379,A -85,B 0,C 180,E1 22872.503,E2 22872.503} C_VEL
LIN {X 0,Y 512.596,Z 610.384,A -85,B 0,C 180,E1 22869.09,E2 22869.09} C_VEL
LIN {X 0,Y 512.629,Z 610.629,A -85,B 0,C 180,E1 22866.915,E2 22866.915} C_VEL
LIN {X 0,Y 515.98,Z 624.52,A -85,B 0,C 180,E1 22865.225,E2 22865.225} C_VEL
LIN {X 0,Y 515.938,Z 651.595,A -85,B 0,C 180,E1 22862.221,E2 22862.221} C_VEL
LIN {X 0,Y 515.674,Z 678.805,A -85,B 0,C 180,E1 22859.111,E2 22859.111} C_VEL
LIN {X 0,Y 515.397,Z 700.47,A -85,B 0,C 180,E1 22856.611,E2 22856.611} C_VEL
LIN {X 0,Y 516.124,Z 706.055,A -85,B 0,C 180,E1 22856.491,E2 22856.491} C_VEL
LIN {X 0,Y 515.209,Z 839.561,A -85,B 0,C 180,E1 22854.519,E2 22854.519} C_VEL
LIN {X 0,Y 515.06,Z 855.37,A -85,B 0,C 180,E1 22854.08,E2 22854.08} C_VEL
LIN {X 0,Y 514.783,Z 871.287,A -85,B 0,C 180,E1 22853.419,E2 22853.419} C_VEL
LIN {X 0,Y 514.444,Z 885.26,A -85,B 0,C 180,E1 22852.63,E2 22852.63} C_VEL
LIN {X 0,Y 514.028,Z 899.164,A -85,B 0,C 180,E1 22851.611,E2 22851.611} C_VEL
LIN {X 0,Y 513.629,Z 911.459,A -85,B 0,C 180,E1 22850.475,E2 22850.475} C_VEL
LIN {X 0,Y 513.199,Z 923.318,A -85,B 0,C 180,E1 22849.095,E2 22849.095} C_VEL
LIN {X 0,Y 512.842,Z 933.351,A -85,B 0,C 180,E1 22847.629,E2 22847.629} C_VEL
LIN {X 0,Y 512.564,Z 942.062,A -85,B 0,C 180,E1 22846.002,E2 22846.002} C_VEL
LIN {X 0,Y 512.38,Z 948.748,A -85,B 0,C 180,E1 22844.378,E2 22844.378} C_VEL
LIN {X 0,Y 512.239,Z 954.301,A -85,B 0,C 180,E1 22842.506,E2 22842.506} C_VEL
LIN {X 0,Y 512.167,Z 957.687,A -85,B 0,C 180,E1 22840.736,E2 22840.736} C_VEL
LIN {X 0,Y 512.135,Z 959.453,A -85,B 0,C 180,E1 22838.827,E2 22838.827} C_VEL
LIN {X 0,Y 512.133,Z 959.374,A -85,B 0,C 180,E1 22837.016,E2 22837.016} C_VEL
LIN {X 0,Y 512.152,Z 957.383,A -85,B 0,C 180,E1 22835.058,E2 22835.058} C_VEL
LIN {X 0,Y 512.16,Z 956.752,A -85,B 0,C 180,E1 22834.683,E2 22834.683} C_VEL
LIN {X 0,Y 511.212,Z 955.242,A -85,B 0,C 180,E1 22833.838,E2 22833.838} C_VEL
LIN {X 0,Y 506.893,Z 952.009,A -85,B 0,C 180,E1 22832.316,E2 22832.316} C_VEL
LIN {X 0,Y 504.801,Z 949.294,A -85,B 0,C 180,E1 22831.381,E2 22831.381} C_VEL
LIN {X 0,Y 504.498,Z 947.579,A -85,B 0,C 180,E1 22830.914,E2 22830.914} C_VEL
LIN {X 0,Y 504.726,Z 940.198,A -85,B 0,C 180,E1 22829.263,E2 22829.263} C_VEL
LIN {X 0,Y 505.035,Z 931.071,A -85,B 0,C 180,E1 22827.687,E2 22827.687} C_VEL
LIN {X 0,Y 505.439,Z 920.492,A -85,B 0,C 180,E1 22826.229,E2 22826.229} C_VEL
LIN {X 0,Y 505.896,Z 908.224,A -85,B 0,C 180,E1 22824.891,E2 22824.891} C_VEL
LIN {X 0,Y 506.35,Z 895.07,A -85,B 0,C 180,E1 22823.743,E2 22823.743} C_VEL
LIN {X 0,Y 506.768,Z 881.221,A -85,B 0,C 180,E1 22822.797,E2 22822.797} C_VEL
LIN {X 0,Y 507.16,Z 866.176,A -85,B 0,C 180,E1 22822.007,E2 22822.007} C_VEL
LIN {X 0,Y 507.426,Z 850.025,A -85,B 0,C 180,E1 22821.406,E2 22821.406} C_VEL
LIN {X 0,Y 507.573,Z 833.555,A -85,B 0,C 180,E1 22821.014,E2 22821.014} C_VEL
LIN {X 0,Y 508.337,Z 704.093,A -85,B 0,C 180,E1 22819.095,E2 22819.095} C_VEL
LIN {X 0,Y 507.277,Z 698.44,A -85,B 0,C 180,E1 22818.932,E2 22818.932} C_VEL
LIN {X 0,Y 507.882,Z 669.181,A -85,B 0,C 180,E1 22815.453,E2 22815.453} C_VEL
LIN {X 0,Y 508.37,Z 640.299,A -85,B 0,C 180,E1 22812.036,E2 22812.036} C_VEL
LIN {X 0,Y 508.418,Z 626.698,A -85,B 0,C 180,E1 22810.44,E2 22810.44} C_VEL
LIN {X 0,Y 504.674,Z 611.527,A -85,B 0,C 180,E1 22808.411,E2 22808.411} C_VEL
LIN {X 0,Y 504.647,Z 611.373,A -85,B 0,C 180,E1 22804.889,E2 22804.889} C_VEL
LIN {X 0,Y 504.71,Z 611.369,A -85,B 0,C 180,E1 22801.534,E2 22801.534} C_VEL
LIN {X 0,Y 504.653,Z 611.369,A -85,B 0,C 180,E1 22798.155,E2 22798.155} C_VEL
LIN {X 0,Y 504.656,Z 611.35,A -85,B 0,C 180,E1 22794.576,E2 22794.576} C_VEL
LIN {X 0,Y 504.709,Z 611.362,A -85,B 0,C 180,E1 22791.256,E2 22791.256} C_VEL
LIN {X 0,Y 504.656,Z 611.372,A -85,B 0,C 180,E1 22787.885,E2 22787.885} C_VEL
LIN {X 0,Y 504.68,Z 611.373,A -85,B 0,C 180,E1 22784.35,E2 22784.35} C_VEL
LIN {X 0,Y 504.716,Z 611.708,A -85,B 0,C 180,E1 22783.487,E2 22783.487} C_VEL
LIN {X 0,Y 509.713,Z 630.183,A -85,B 0,C 180,E1 22780.626,E2 22780.626} C_VEL
LIN {X 0,Y 508.587,Z 656.234,A -85,B 0,C 180,E1 22777.228,E2 22777.228} C_VEL
LIN {X 0,Y 507.494,Z 683.369,A -85,B 0,C 180,E1 22773.728,E2 22773.728} C_VEL
LIN {X 0,Y 507.204,Z 693.359,A -85,B 0,C 180,E1 22772.486,E2 22772.486} C_VEL
LIN {X 0,Y 509.739,Z 706.736,A -85,B 0,C 180,E1 22772.133,E2 22772.133} C_VEL
LIN {X 0,Y 508.649,Z 837.036,A -85,B 0,C 180,E1 22770.197,E2 22770.197} C_VEL
LIN {X 0,Y 508.361,Z 853.994,A -85,B 0,C 180,E1 22769.719,E2 22769.719} C_VEL
LIN {X 0,Y 507.972,Z 868.85,A -85,B 0,C 180,E1 22769.098,E2 22769.098} C_VEL
LIN {X 0,Y 507.441,Z 883.757,A -85,B 0,C 180,E1 22768.25,E2 22768.25} C_VEL
LIN {X 0,Y 506.862,Z 897.7,A -85,B 0,C 180,E1 22767.23,E2 22767.23} C_VEL
LIN {X 0,Y 506.284,Z 910.565,A -85,B 0,C 180,E1 22766.037,E2 22766.037} C_VEL
LIN {X 0,Y 505.722,Z 922.376,A -85,B 0,C 180,E1 22764.668,E2 22764.668} C_VEL
LIN {X 0,Y 505.233,Z 932.682,A -85,B 0,C 180,E1 22763.181,E2 22763.181} C_VEL
LIN {X 0,Y 504.84,Z 941.477,A -85,B 0,C 180,E1 22761.573,E2 22761.573} C_VEL
LIN {X 0,Y 504.57,Z 948.847,A -85,B 0,C 180,E1 22759.842,E2 22759.842} C_VEL
LIN {X 0,Y 504.391,Z 954.584,A -85,B 0,C 180,E1 22757.987,E2 22757.987} C_VEL
LIN {X 0,Y 504.29,Z 958.49,A -85,B 0,C 180,E1 22756.119,E2 22756.119} C_VEL
LIN {X 0,Y 504.241,Z 960.549,A -85,B 0,C 180,E1 22754.237,E2 22754.237} C_VEL
LIN {X 0,Y 504.24,Z 960.9,A -85,B 0,C 180,E1 22752.339,E2 22752.339} C_VEL
LIN {X 0,Y 504.276,Z 959.609,A -85,B 0,C 180,E1 22750.543,E2 22750.543} C_VEL
LIN {X 0,Y 504.367,Z 956.364,A -85,B 0,C 180,E1 22748.607,E2 22748.607} C_VEL
LIN {X 0,Y 504.526,Z 951.486,A -85,B 0,C 180,E1 22746.773,E2 22746.773} C_VEL
LIN {X 0,Y 504.758,Z 944.997,A -85,B 0,C 180,E1 22745.044,E2 22745.044} C_VEL
LIN {X 0,Y 505.109,Z 937.105,A -85,B 0,C 180,E1 22743.426,E2 22743.426} C_VEL
LIN {X 0,Y 505.571,Z 927.594,A -85,B 0,C 180,E1 22741.891,E2 22741.891} C_VEL
LIN {X 0,Y 506.147,Z 916.014,A -85,B 0,C 180,E1 22740.406,E2 22740.406} C_VEL
LIN {X 0,Y 506.742,Z 903.612,A -85,B 0,C 180,E1 22739.136,E2 22739.136} C_VEL
LIN {X 0,Y 507.365,Z 889.407,A -85,B 0,C 180,E1 22737.987,E2 22737.987} C_VEL
LIN {X 0,Y 507.912,Z 875.219,A -85,B 0,C 180,E1 22737.09,E2 22737.09} C_VEL
LIN {X 0,Y 508.391,Z 859.533,A -85,B 0,C 180,E1 22736.35,E2 22736.35} C_VEL
LIN {X 0,Y 508.733,Z 843.265,A -85,B 0,C 180,E1 22735.81,E2 22735.81} C_VEL
LIN {X 0,Y 508.917,Z 825.252,A -85,B 0,C 180,E1 22735.464,E2 22735.464} C_VEL
LIN {X 0,Y 509.787,Z 704.872,A -85,B 0,C 180,E1 22733.675,E2 22733.675} C_VEL
LIN {X 0,Y 507.424,Z 693.852,A -85,B 0,C 180,E1 22733.362,E2 22733.362} C_VEL
LIN {X 0,Y 507.734,Z 683.565,A -85,B 0,C 180,E1 22732.091,E2 22732.091} C_VEL
LIN {X 0,Y 508.912,Z 656.244,A -85,B 0,C 180,E1 22728.54,E2 22728.54} C_VEL
LIN {X 0,Y 510.136,Z 630.971,A -85,B 0,C 180,E1 22725.196,E2 22725.196} C_VEL
LIN {X 0,Y 505.35,Z 613.717,A -85,B 0,C 180,E1 22722.43,E2 22722.43} C_VEL
LIN {X 0,Y 504.717,Z 611.456,A -85,B 0,C 180,E1 22721.992,E2 22721.992} C_VEL
LIN {X 0,Y 504.699,Z 611.367,A -85,B 0,C 180,E1 22718.468,E2 22718.468} C_VEL
LIN {X 0,Y 504.694,Z 611.368,A -85,B 0,C 180,E1 22715.067,E2 22715.067} C_VEL
LIN {X 0,Y 504.705,Z 611.359,A -85,B 0,C 180,E1 22711.534,E2 22711.534} C_VEL
LIN {X 0,Y 504.696,Z 611.369,A -85,B 0,C 180,E1 22707.924,E2 22707.924} C_VEL
LIN {X 0,Y 504.699,Z 611.364,A -85,B 0,C 180,E1 22704.46,E2 22704.46} C_VEL
LIN {X 0,Y 504.709,Z 611.362,A -85,B 0,C 180,E1 22700.891,E2 22700.891} C_VEL
LIN {X 0,Y 504.693,Z 611.368,A -85,B 0,C 180,E1 22697.407,E2 22697.407} C_VEL
LIN {X 0,Y 504.703,Z 611.36,A -85,B 0,C 180,E1 22693.87,E2 22693.87} C_VEL
LIN {X 0,Y 504.702,Z 611.358,A -85,B 0,C 180,E1 22690.271,E2 22690.271} C_VEL
LIN {X 0,Y 504.688,Z 611.363,A -85,B 0,C 180,E1 22686.827,E2 22686.827} C_VEL
LIN {X 0,Y 504.704,Z 611.37,A -85,B 0,C 180,E1 22683.294,E2 22683.294} C_VEL
LIN {X 0,Y 504.703,Z 611.357,A -85,B 0,C 180,E1 22679.773,E2 22679.773} C_VEL
LIN {X 0,Y 504.687,Z 611.355,A -85,B 0,C 180,E1 22676.252,E2 22676.252} C_VEL
LIN {X 0,Y 504.702,Z 611.365,A -85,B 0,C 180,E1 22672.716,E2 22672.716} C_VEL
LIN {X 0,Y 504.701,Z 611.362,A -85,B 0,C 180,E1 22669.152,E2 22669.152} C_VEL
LIN {X 0,Y 504.691,Z 611.357,A -85,B 0,C 180,E1 22665.643,E2 22665.643} C_VEL
LIN {X 0,Y 504.69,Z 611.36,A -85,B 0,C 180,E1 22662.117,E2 22662.117} C_VEL
LIN {X 0,Y 504.703,Z 611.367,A -85,B 0,C 180,E1 22658.608,E2 22658.608} C_VEL
LIN {X 0,Y 504.693,Z 611.364,A -85,B 0,C 180,E1 22655.142,E2 22655.142} C_VEL
LIN {X 0,Y 504.687,Z 611.369,A -85,B 0,C 180,E1 22651.597,E2 22651.597} C_VEL
LIN {X 0,Y 504.707,Z 611.359,A -85,B 0,C 180,E1 22648.198,E2 22648.198} C_VEL
LIN {X 0,Y 504.693,Z 611.361,A -85,B 0,C 180,E1 22644.656,E2 22644.656} C_VEL
LIN {X 0,Y 504.682,Z 611.37,A -85,B 0,C 180,E1 22641.095,E2 22641.095} C_VEL
LIN {X 0,Y 504.708,Z 611.368,A -85,B 0,C 180,E1 22637.641,E2 22637.641} C_VEL
LIN {X 0,Y 504.693,Z 611.364,A -85,B 0,C 180,E1 22634.179,E2 22634.179} C_VEL
LIN {X 0,Y 504.68,Z 611.37,A -85,B 0,C 180,E1 22630.643,E2 22630.643} C_VEL
LIN {X 0,Y 504.708,Z 611.369,A -85,B 0,C 180,E1 22627.173,E2 22627.173} C_VEL
LIN {X 0,Y 504.741,Z 611.78,A -85,B 0,C 180,E1 22626.505,E2 22626.505} C_VEL
LIN {X 0,Y 511.845,Z 631.853,A -85,B 0,C 180,E1 22624.18,E2 22624.18} C_VEL
LIN {X 0,Y 513.715,Z 637.665,A -85,B 0,C 180,E1 22623.556,E2 22623.556} C_VEL
LIN {X 0,Y 511.968,Z 680.767,A -85,B 0,C 180,E1 22620.062,E2 22620.062} C_VEL
LIN {X 0,Y 510.982,Z 709.594,A -85,B 0,C 180,E1 22617.809,E2 22617.809} C_VEL
LIN {X 0,Y 513.334,Z 725.798,A -85,B 0,C 180,E1 22617.452,E2 22617.452} C_VEL
LIN {X 0,Y 511.621,Z 927.16,A -85,B 0,C 180,E1 22614.533,E2 22614.533} C_VEL
LIN {X 0,Y 511.086,Z 946.631,A -85,B 0,C 180,E1 22614.038,E2 22614.038} C_VEL
LIN {X 0,Y 510.391,Z 965.395,A -85,B 0,C 180,E1 22613.343,E2 22613.343} C_VEL
LIN {X 0,Y 509.588,Z 983.364,A -85,B 0,C 180,E1 22612.46,E2 22612.46} C_VEL
LIN {X 0,Y 508.693,Z 1000.698,A -85,B 0,C 180,E1 22611.383,E2 22611.383} C_VEL
LIN {X 0,Y 507.801,Z 1016.785,A -85,B 0,C 180,E1 22610.156,E2 22610.156} C_VEL
LIN {X 0,Y 506.886,Z 1032.542,A -85,B 0,C 180,E1 22608.695,E2 22608.695} C_VEL
LIN {X 0,Y 506.08,Z 1046.684,A -85,B 0,C 180,E1 22607.12,E2 22607.12} C_VEL
LIN {X 0,Y 505.38,Z 1059.758,A -85,B 0,C 180,E1 22605.373,E2 22605.373} C_VEL
LIN {X 0,Y 504.816,Z 1071.553,A -85,B 0,C 180,E1 22603.47,E2 22603.47} C_VEL
LIN {X 0,Y 504.419,Z 1081.34,A -85,B 0,C 180,E1 22601.549,E2 22601.549} C_VEL
LIN {X 0,Y 504.164,Z 1089.434,A -85,B 0,C 180,E1 22599.589,E2 22599.589} C_VEL
LIN {X 0,Y 504.006,Z 1096.129,A -85,B 0,C 180,E1 22597.523,E2 22597.523} C_VEL
LIN {X 0,Y 503.932,Z 1101.294,A -85,B 0,C 180,E1 22595.351,E2 22595.351} C_VEL
LIN {X 0,Y 503.913,Z 1104.657,A -85,B 0,C 180,E1 22593.185,E2 22593.185} C_VEL
LIN {X 0,Y 503.908,Z 1106.303,A -85,B 0,C 180,E1 22591.023,E2 22591.023} C_VEL
LIN {X 0,Y 503.906,Z 1106.265,A -85,B 0,C 180,E1 22588.863,E2 22588.863} C_VEL
LIN {X 0,Y 503.914,Z 1104.539,A -85,B 0,C 180,E1 22586.701,E2 22586.701} C_VEL
LIN {X 0,Y 503.936,Z 1101.085,A -85,B 0,C 180,E1 22584.535,E2 22584.535} C_VEL
LIN {X 0,Y 504.012,Z 1095.817,A -85,B 0,C 180,E1 22582.362,E2 22582.362} C_VEL
LIN {X 0,Y 504.189,Z 1088.59,A -85,B 0,C 180,E1 22580.18,E2 22580.18} C_VEL
LIN {X 0,Y 504.48,Z 1079.732,A -85,B 0,C 180,E1 22578.104,E2 22578.104} C_VEL
LIN {X 0,Y 504.914,Z 1069.305,A -85,B 0,C 180,E1 22576.136,E2 22576.136} C_VEL
LIN {X 0,Y 505.46,Z 1058.165,A -85,B 0,C 180,E1 22574.393,E2 22574.393} C_VEL
LIN {X 0,Y 506.188,Z 1044.739,A -85,B 0,C 180,E1 22572.646,E2 22572.646} C_VEL
LIN {X 0,Y 507.019,Z 1030.196,A -85,B 0,C 180,E1 22571.07,E2 22571.07} C_VEL
LIN {X 0,Y 507.914,Z 1014.628,A -85,B 0,C 180,E1 22569.668,E2 22569.668} C_VEL
LIN {X 0,Y 508.826,Z 998.081,A -85,B 0,C 180,E1 22568.441,E2 22568.441} C_VEL
LIN {X 0,Y 509.721,Z 980.552,A -85,B 0,C 180,E1 22567.389,E2 22567.389} C_VEL
LIN {X 0,Y 510.508,Z 962.6,A -85,B 0,C 180,E1 22566.542,E2 22566.542} C_VEL
LIN {X 0,Y 511.15,Z 944.087,A -85,B 0,C 180,E1 22565.887,E2 22565.887} C_VEL
LIN {X 0,Y 511.647,Z 925.16,A -85,B 0,C 180,E1 22565.431,E2 22565.431} C_VEL
LIN {X 0,Y 513.195,Z 723.345,A -85,B 0,C 180,E1 22562.5,E2 22562.5} C_VEL
LIN {X 0,Y 510.966,Z 708.785,A -85,B 0,C 180,E1 22562.145,E2 22562.145} C_VEL
LIN {X 0,Y 512.54,Z 665.375,A -85,B 0,C 180,E1 22558.699,E2 22558.699} C_VEL
LIN {X 0,Y 513.71,Z 636.908,A -85,B 0,C 180,E1 22556.361,E2 22556.361} C_VEL
LIN {X 0,Y 505.141,Z 613.221,A -85,B 0,C 180,E1 22553.668,E2 22553.668} C_VEL
LIN {X 0,Y 504.716,Z 611.566,A -85,B 0,C 180,E1 22553.434,E2 22553.434} C_VEL
LIN {X 0,Y 504.693,Z 611.367,A -85,B 0,C 180,E1 22549.919,E2 22549.919} C_VEL
LIN {X 0,Y 504.702,Z 611.363,A -85,B 0,C 180,E1 22546.415,E2 22546.415} C_VEL
LIN {X 0,Y 504.705,Z 611.371,A -85,B 0,C 180,E1 22542.805,E2 22542.805} C_VEL
LIN {X 0,Y 504.697,Z 611.367,A -85,B 0,C 180,E1 22539.342,E2 22539.342} C_VEL
LIN {X 0,Y 504.696,Z 611.365,A -85,B 0,C 180,E1 22535.877,E2 22535.877} C_VEL
LIN {X 0,Y 504.695,Z 611.37,A -85,B 0,C 180,E1 22532.337,E2 22532.337} C_VEL
LIN {X 0,Y 504.706,Z 611.366,A -85,B 0,C 180,E1 22528.879,E2 22528.879} C_VEL
LIN {X 0,Y 504.695,Z 611.365,A -85,B 0,C 180,E1 22525.336,E2 22525.336} C_VEL
LIN {X 0,Y 504.679,Z 611.37,A -85,B 0,C 180,E1 22521.867,E2 22521.867} C_VEL
LIN {X 0,Y 504.709,Z 611.369,A -85,B 0,C 180,E1 22518.36,E2 22518.36} C_VEL
LIN {X 0,Y 504.682,Z 611.368,A -85,B 0,C 180,E1 22514.925,E2 22514.925} C_VEL
LIN {X 0,Y 504.662,Z 611.373,A -85,B 0,C 180,E1 22511.427,E2 22511.427} C_VEL
LIN {X 0,Y 504.708,Z 611.369,A -85,B 0,C 180,E1 22507.971,E2 22507.971} C_VEL
LIN {X 0,Y 504.7,Z 611.682,A -85,B 0,C 180,E1 22507.241,E2 22507.241} C_VEL
LIN {X 0,Y 508.399,Z 626.526,A -85,B 0,C 180,E1 22505.417,E2 22505.417} C_VEL
LIN {X 0,Y 508.404,Z 653.191,A -85,B 0,C 180,E1 22502.468,E2 22502.468} C_VEL
LIN {X 0,Y 508.101,Z 682.639,A -85,B 0,C 180,E1 22499.098,E2 22499.098} C_VEL
LIN {X 0,Y 507.872,Z 701.825,A -85,B 0,C 180,E1 22496.889,E2 22496.889} C_VEL
LIN {X 0,Y 508.557,Z 706.96,A -85,B 0,C 180,E1 22496.772,E2 22496.772} C_VEL
LIN {X 0,Y 507.528,Z 840.965,A -85,B 0,C 180,E1 22494.747,E2 22494.747} C_VEL
LIN {X 0,Y 507.384,Z 856.79,A -85,B 0,C 180,E1 22494.3,E2 22494.3} C_VEL
LIN {X 0,Y 507.113,Z 872.024,A -85,B 0,C 180,E1 22493.661,E2 22493.661} C_VEL
LIN {X 0,Y 506.763,Z 886.165,A -85,B 0,C 180,E1 22492.859,E2 22492.859} C_VEL
LIN {X 0,Y 506.321,Z 900.148,A -85,B 0,C 180,E1 22491.826,E2 22491.826} C_VEL
LIN {X 0,Y 505.895,Z 912.524,A -85,B 0,C 180,E1 22490.673,E2 22490.673} C_VEL
LIN {X 0,Y 505.431,Z 924.343,A -85,B 0,C 180,E1 22489.283,E2 22489.283} C_VEL
LIN {X 0,Y 505.065,Z 933.893,A -85,B 0,C 180,E1 22487.887,E2 22487.887} C_VEL
LIN {X 0,Y 504.742,Z 942.685,A -85,B 0,C 180,E1 22486.248,E2 22486.248} C_VEL
LIN {X 0,Y 504.534,Z 949.54,A -85,B 0,C 180,E1 22484.6,E2 22484.6} C_VEL
LIN {X 0,Y 504.366,Z 954.92,A -85,B 0,C 180,E1 22482.819,E2 22482.819} C_VEL
LIN {X 0,Y 504.279,Z 958.561,A -85,B 0,C 180,E1 22481.024,E2 22481.024} C_VEL
LIN {X 0,Y 504.236,Z 960.47,A -85,B 0,C 180,E1 22479.21,E2 22479.21} C_VEL
LIN {X 0,Y 504.222,Z 960.696,A -85,B 0,C 180,E1 22477.252,E2 22477.252} C_VEL
LIN {X 0,Y 504.238,Z 959.075,A -85,B 0,C 180,E1 22475.391,E2 22475.391} C_VEL
LIN {X 0,Y 504.299,Z 955.647,A -85,B 0,C 180,E1 22473.506,E2 22473.506} C_VEL
LIN {X 0,Y 504.417,Z 950.526,A -85,B 0,C 180,E1 22471.722,E2 22471.722} C_VEL
LIN {X 0,Y 504.498,Z 947.579,A -85,B 0,C 180,E1 22470.914,E2 22470.914} C_VEL
LIN {X 0,Y 503.61,Z 944.452,A -85,B 0,C 180,E1 22470.113,E2 22470.113} C_VEL
LIN {X 0,Y 499.135,Z 937.845,A -85,B 0,C 180,E1 22468.574,E2 22468.574} C_VEL
LIN {X 0,Y 497.367,Z 933.282,A -85,B 0,C 180,E1 22467.717,E2 22467.717} C_VEL
LIN {X 0,Y 497.253,Z 931.316,A -85,B 0,C 180,E1 22467.404,E2 22467.404} C_VEL
LIN {X 0,Y 497.681,Z 920.818,A -85,B 0,C 180,E1 22465.968,E2 22465.968} C_VEL
LIN {X 0,Y 498.199,Z 907.974,A -85,B 0,C 180,E1 22464.57,E2 22464.57} C_VEL
LIN {X 0,Y 498.663,Z 894.978,A -85,B 0,C 180,E1 22463.451,E2 22463.451} C_VEL
LIN {X 0,Y 499.14,Z 880.079,A -85,B 0,C 180,E1 22462.445,E2 22462.445} C_VEL
LIN {X 0,Y 499.52,Z 865.165,A -85,B 0,C 180,E1 22461.688,E2 22461.688} C_VEL
LIN {X 0,Y 499.8,Z 848.541,A -85,B 0,C 180,E1 22461.088,E2 22461.088} C_VEL
LIN {X 0,Y 499.914,Z 831.532,A -85,B 0,C 180,E1 22460.719,E2 22460.719} C_VEL
LIN {X 0,Y 500.767,Z 705.2,A -85,B 0,C 180,E1 22458.812,E2 22458.812} C_VEL
LIN {X 0,Y 499.676,Z 699.414,A -85,B 0,C 180,E1 22458.645,E2 22458.645} C_VEL
LIN {X 0,Y 500.304,Z 669.99,A -85,B 0,C 180,E1 22455.132,E2 22455.132} C_VEL
LIN {X 0,Y 500.79,Z 641.274,A -85,B 0,C 180,E1 22451.741,E2 22451.741} C_VEL
LIN {X 0,Y 500.759,Z 628.612,A -85,B 0,C 180,E1 22450.236,E2 22450.236} C_VEL
LIN {X 0,Y 496.764,Z 612.51,A -85,B 0,C 180,E1 22448.073,E2 22448.073} C_VEL
LIN {X 0,Y 496.705,Z 612.363,A -85,B 0,C 180,E1 22444.728,E2 22444.728} C_VEL
LIN {X 0,Y 496.752,Z 612.356,A -85,B 0,C 180,E1 22441.286,E2 22441.286} C_VEL
LIN {X 0,Y 496.727,Z 612.359,A -85,B 0,C 180,E1 22437.912,E2 22437.912} C_VEL
LIN {X 0,Y 496.711,Z 612.339,A -85,B 0,C 180,E1 22434.372,E2 22434.372} C_VEL
LIN {X 0,Y 496.765,Z 612.346,A -85,B 0,C 180,E1 22430.946,E2 22430.946} C_VEL
LIN {X 0,Y 496.738,Z 612.361,A -85,B 0,C 180,E1 22427.453,E2 22427.453} C_VEL
LIN {X 0,Y 496.739,Z 612.495,A -85,B 0,C 180,E1 22423.975,E2 22423.975} C_VEL
LIN {X 0,Y 501.637,Z 630.293,A -85,B 0,C 180,E1 22421.148,E2 22421.148} C_VEL
LIN {X 0,Y 502.186,Z 633.515,A -85,B 0,C 180,E1 22420.671,E2 22420.671} C_VEL
LIN {X 0,Y 500.938,Z 660.63,A -85,B 0,C 180,E1 22417.109,E2 22417.109} C_VEL
LIN {X 0,Y 499.697,Z 688.724,A -85,B 0,C 180,E1 22413.442,E2 22413.442} C_VEL
LIN {X 0,Y 499.621,Z 693.787,A -85,B 0,C 180,E1 22412.839,E2 22412.839} C_VEL
LIN {X 0,Y 502.365,Z 707.951,A -85,B 0,C 180,E1 22412.471,E2 22412.471} C_VEL
LIN {X 0,Y 501.187,Z 837.623,A -85,B 0,C 180,E1 22410.518,E2 22410.518} C_VEL
LIN {X 0,Y 500.883,Z 854.538,A -85,B 0,C 180,E1 22410.036,E2 22410.036} C_VEL
LIN {X 0,Y 500.443,Z 870.188,A -85,B 0,C 180,E1 22409.371,E2 22409.371} C_VEL
LIN {X 0,Y 499.875,Z 885.008,A -85,B 0,C 180,E1 22408.51,E2 22408.51} C_VEL
LIN {X 0,Y 499.252,Z 898.905,A -85,B 0,C 180,E1 22407.475,E2 22407.475} C_VEL
LIN {X 0,Y 498.619,Z 911.724,A -85,B 0,C 180,E1 22406.264,E2 22406.264} C_VEL
LIN {X 0,Y 497.979,Z 924.066,A -85,B 0,C 180,E1 22404.804,E2 22404.804} C_VEL
LIN {X 0,Y 497.444,Z 934.153,A -85,B 0,C 180,E1 22403.306,E2 22403.306} C_VEL
LIN {X 0,Y 496.992,Z 943.447,A -85,B 0,C 180,E1 22401.555,E2 22401.555} C_VEL
LIN {X 0,Y 496.687,Z 950.585,A -85,B 0,C 180,E1 22399.797,E2 22399.797} C_VEL
LIN {X 0,Y 496.497,Z 956.173,A -85,B 0,C 180,E1 22397.911,E2 22397.911} C_VEL
LIN {X 0,Y 496.378,Z 959.903,A -85,B 0,C 180,E1 22396.012,E2 22396.012} C_VEL
LIN {X 0,Y 496.329,Z 961.898,A -85,B 0,C 180,E1 22393.979,E2 22393.979} C_VEL
LIN {X 0,Y 496.333,Z 962.003,A -85,B 0,C 180,E1 22392.048,E2 22392.048} C_VEL
LIN {X 0,Y 496.386,Z 960.285,A -85,B 0,C 180,E1 22390.098,E2 22390.098} C_VEL
LIN {X 0,Y 496.513,Z 956.823,A -85,B 0,C 180,E1 22388.179,E2 22388.179} C_VEL
LIN {X 0,Y 496.712,Z 951.356,A -85,B 0,C 180,E1 22386.26,E2 22386.26} C_VEL
LIN {X 0,Y 497.026,Z 944.498,A -85,B 0,C 180,E1 22384.501,E2 22384.501} C_VEL
LIN {X 0,Y 497.445,Z 936.065,A -85,B 0,C 180,E1 22382.854,E2 22382.854} C_VEL
LIN {X 0,Y 498.021,Z 925.773,A -85,B 0,C 180,E1 22381.26,E2 22381.26} C_VEL
LIN {X 0,Y 498.643,Z 914.224,A -85,B 0,C 180,E1 22379.842,E2 22379.842} C_VEL
LIN {X 0,Y 499.329,Z 901.004,A -85,B 0,C 180,E1 22378.543,E2 22378.543} C_VEL
LIN {X 0,Y 499.946,Z 887.899,A -85,B 0,C 180,E1 22377.522,E2 22377.522} C_VEL
LIN {X 0,Y 500.545,Z 872.899,A -85,B 0,C 180,E1 22376.614,E2 22376.614} C_VEL
LIN {X 0,Y 501.039,Z 857.4,A -85,B 0,C 180,E1 22375.911,E2 22375.911} C_VEL
LIN {X 0,Y 501.352,Z 840.989,A -85,B 0,C 180,E1 22375.409,E2 22375.409} C_VEL
LIN {X 0,Y 501.588,Z 817.581,A -85,B 0,C 180,E1 22375.002,E2 22375.002} C_VEL
LIN {X 0,Y 502.492,Z 706.174,A -85,B 0,C 180,E1 22373.318,E2 22373.318} C_VEL
LIN {X 0,Y 499.858,Z 693.792,A -85,B 0,C 180,E1 22372.951,E2 22372.951} C_VEL
LIN {X 0,Y 500.993,Z 666.474,A -85,B 0,C 180,E1 22369.412,E2 22369.412} C_VEL
LIN {X 0,Y 502.398,Z 639.741,A -85,B 0,C 180,E1 22365.849,E2 22365.849} C_VEL
LIN {X 0,Y 502.554,Z 633.06,A -85,B 0,C 180,E1 22364.935,E2 22364.935} C_VEL
LIN {X 0,Y 498.275,Z 617.526,A -85,B 0,C 180,E1 22362.395,E2 22362.395} C_VEL
LIN {X 0,Y 496.766,Z 612.438,A -85,B 0,C 180,E1 22361.468,E2 22361.468} C_VEL
LIN {X 0,Y 496.758,Z 612.354,A -85,B 0,C 180,E1 22358.018,E2 22358.018} C_VEL
LIN {X 0,Y 496.762,Z 612.355,A -85,B 0,C 180,E1 22354.389,E2 22354.389} C_VEL
LIN {X 0,Y 496.755,Z 612.351,A -85,B 0,C 180,E1 22350.881,E2 22350.881} C_VEL
LIN {X 0,Y 496.765,Z 612.353,A -85,B 0,C 180,E1 22347.317,E2 22347.317} C_VEL
LIN {X 0,Y 496.755,Z 612.356,A -85,B 0,C 180,E1 22343.679,E2 22343.679} C_VEL
LIN {X 0,Y 496.765,Z 612.358,A -85,B 0,C 180,E1 22340.132,E2 22340.132} C_VEL
LIN {X 0,Y 496.763,Z 612.353,A -85,B 0,C 180,E1 22336.487,E2 22336.487} C_VEL
LIN {X 0,Y 496.752,Z 612.355,A -85,B 0,C 180,E1 22333.029,E2 22333.029} C_VEL
LIN {X 0,Y 496.764,Z 612.349,A -85,B 0,C 180,E1 22329.5,E2 22329.5} C_VEL
LIN {X 0,Y 496.763,Z 612.349,A -85,B 0,C 180,E1 22326.008,E2 22326.008} C_VEL
LIN {X 0,Y 496.754,Z 612.352,A -85,B 0,C 180,E1 22322.423,E2 22322.423} C_VEL
LIN {X 0,Y 496.758,Z 612.358,A -85,B 0,C 180,E1 22318.847,E2 22318.847} C_VEL
LIN {X 0,Y 496.761,Z 612.344,A -85,B 0,C 180,E1 22315.267,E2 22315.267} C_VEL
LIN {X 0,Y 496.767,Z 612.346,A -85,B 0,C 180,E1 22311.668,E2 22311.668} C_VEL
LIN {X 0,Y 496.747,Z 612.355,A -85,B 0,C 180,E1 22308.153,E2 22308.153} C_VEL
LIN {X 0,Y 496.768,Z 612.352,A -85,B 0,C 180,E1 22304.593,E2 22304.593} C_VEL
LIN {X 0,Y 496.766,Z 612.342,A -85,B 0,C 180,E1 22300.97,E2 22300.97} C_VEL
LIN {X 0,Y 496.744,Z 612.348,A -85,B 0,C 180,E1 22297.5,E2 22297.5} C_VEL
LIN {X 0,Y 496.761,Z 612.355,A -85,B 0,C 180,E1 22293.974,E2 22293.974} C_VEL
LIN {X 0,Y 496.768,Z 612.355,A -85,B 0,C 180,E1 22290.4,E2 22290.4} C_VEL
LIN {X 0,Y 496.75,Z 612.355,A -85,B 0,C 180,E1 22286.858,E2 22286.858} C_VEL
LIN {X 0,Y 496.746,Z 612.357,A -85,B 0,C 180,E1 22283.235,E2 22283.235} C_VEL
LIN {X 0,Y 496.769,Z 612.356,A -85,B 0,C 180,E1 22279.713,E2 22279.713} C_VEL
LIN {X 0,Y 496.765,Z 612.349,A -85,B 0,C 180,E1 22276.101,E2 22276.101} C_VEL
LIN {X 0,Y 496.738,Z 612.358,A -85,B 0,C 180,E1 22272.549,E2 22272.549} C_VEL
LIN {X 0,Y 496.77,Z 612.358,A -85,B 0,C 180,E1 22269.048,E2 22269.048} C_VEL
LIN {X 0,Y 496.806,Z 612.627,A -85,B 0,C 180,E1 22267.068,E2 22267.068} C_VEL
LIN {X 0,Y 503.23,Z 630.879,A -85,B 0,C 180,E1 22264.857,E2 22264.857} C_VEL
LIN {X 0,Y 506.422,Z 639.933,A -85,B 0,C 180,E1 22263.832,E2 22263.832} C_VEL
LIN {X 0,Y 504.394,Z 684.367,A -85,B 0,C 180,E1 22260.166,E2 22260.166} C_VEL
LIN {X 0,Y 503.463,Z 709.124,A -85,B 0,C 180,E1 22258.192,E2 22258.192} C_VEL
LIN {X 0,Y 505.962,Z 726.984,A -85,B 0,C 180,E1 22257.789,E2 22257.789} C_VEL
LIN {X 0,Y 504.114,Z 926.829,A -85,B 0,C 180,E1 22254.852,E2 22254.852} C_VEL
LIN {X 0,Y 503.556,Z 946.575,A -85,B 0,C 180,E1 22254.35,E2 22254.35} C_VEL
LIN {X 0,Y 502.854,Z 965.6,A -85,B 0,C 180,E1 22253.65,E2 22253.65} C_VEL
LIN {X 0,Y 502.056,Z 983.725,A -85,B 0,C 180,E1 22252.768,E2 22252.768} C_VEL
LIN {X 0,Y 501.22,Z 999.86,A -85,B 0,C 180,E1 22251.78,E2 22251.78} C_VEL
LIN {X 0,Y 500.195,Z 1016.783,A -85,B 0,C 180,E1 22250.476,E2 22250.476} C_VEL
LIN {X 0,Y 499.224,Z 1032.179,A -85,B 0,C 180,E1 22249.033,E2 22249.033} C_VEL
LIN {X 0,Y 498.311,Z 1046.684,A -85,B 0,C 180,E1 22247.395,E2 22247.395} C_VEL
LIN {X 0,Y 497.542,Z 1059.758,A -85,B 0,C 180,E1 22245.622,E2 22245.622} C_VEL
LIN {X 0,Y 496.929,Z 1071.302,A -85,B 0,C 180,E1 22243.734,E2 22243.734} C_VEL
LIN {X 0,Y 496.478,Z 1081.339,A -85,B 0,C 180,E1 22241.736,E2 22241.736} C_VEL
LIN {X 0,Y 496.196,Z 1089.434,A -85,B 0,C 180,E1 22239.745,E2 22239.745} C_VEL
LIN {X 0,Y 496.018,Z 1096.129,A -85,B 0,C 180,E1 22237.645,E2 22237.645} C_VEL
LIN {X 0,Y 495.936,Z 1101.294,A -85,B 0,C 180,E1 22235.437,E2 22235.437} C_VEL
LIN {X 0,Y 495.914,Z 1104.656,A -85,B 0,C 180,E1 22233.236,E2 22233.236} C_VEL
LIN {X 0,Y 495.907,Z 1106.303,A -85,B 0,C 180,E1 22231.039,E2 22231.039} C_VEL
LIN {X 0,Y 495.906,Z 1106.266,A -85,B 0,C 180,E1 22228.844,E2 22228.844} C_VEL
LIN {X 0,Y 495.913,Z 1104.539,A -85,B 0,C 180,E1 22226.648,E2 22226.648} C_VEL
LIN {X 0,Y 495.941,Z 1101.085,A -85,B 0,C 180,E1 22224.446,E2 22224.446} C_VEL
LIN {X 0,Y 496.027,Z 1095.817,A -85,B 0,C 180,E1 22222.238,E2 22222.238} C_VEL
LIN {X 0,Y 496.209,Z 1089.024,A -85,B 0,C 180,E1 22220.138,E2 22220.138} C_VEL
LIN {X 0,Y 496.526,Z 1080.297,A -85,B 0,C 180,E1 22218.029,E2 22218.029} C_VEL
LIN {X 0,Y 496.997,Z 1070.003,A -85,B 0,C 180,E1 22216.03,E2 22216.03} C_VEL
LIN {X 0,Y 497.632,Z 1058.164,A -85,B 0,C 180,E1 22214.142,E2 22214.142} C_VEL
LIN {X 0,Y 498.439,Z 1044.739,A -85,B 0,C 180,E1 22212.368,E2 22212.368} C_VEL
LIN {X 0,Y 499.348,Z 1030.195,A -85,B 0,C 180,E1 22210.768,E2 22210.768} C_VEL
LIN {X 0,Y 500.324,Z 1014.625,A -85,B 0,C 180,E1 22209.346,E2 22209.346} C_VEL
LIN {X 0,Y 501.266,Z 998.959,A -85,B 0,C 180,E1 22208.16,E2 22208.16} C_VEL
LIN {X 0,Y 502.136,Z 982.312,A -85,B 0,C 180,E1 22207.152,E2 22207.152} C_VEL
LIN {X 0,Y 502.944,Z 963.865,A -85,B 0,C 180,E1 22206.273,E2 22206.273} C_VEL
LIN {X 0,Y 503.634,Z 944.278,A -85,B 0,C 180,E1 22205.577,E2 22205.577} C_VEL
LIN {X 0,Y 504.156,Z 924.739,A -85,B 0,C 180,E1 22205.106,E2 22205.106} C_VEL
LIN {X 0,Y 505.832,Z 724.374,A -85,B 0,C 180,E1 22202.156,E2 22202.156} C_VEL
LIN {X 0,Y 503.487,Z 709.048,A -85,B 0,C 180,E1 22201.794,E2 22201.794} C_VEL
LIN {X 0,Y 505.211,Z 666.044,A -85,B 0,C 180,E1 22198.321,E2 22198.321} C_VEL
LIN {X 0,Y 506.436,Z 639.781,A -85,B 0,C 180,E1 22196.129,E2 22196.129} C_VEL
LIN {X 0,Y 497.649,Z 615.194,A -85,B 0,C 180,E1 22193.288,E2 22193.288} C_VEL
LIN {X 0,Y 496.795,Z 612.564,A -85,B 0,C 180,E1 22192.93,E2 22192.93} C_VEL
LIN {X 0,Y 496.75,Z 612.356,A -85,B 0,C 180,E1 22189.448,E2 22189.448} C_VEL
LIN {X 0,Y 496.763,Z 612.35,A -85,B 0,C 180,E1 22185.86,E2 22185.86} C_VEL
LIN {X 0,Y 496.759,Z 612.355,A -85,B 0,C 180,E1 22182.38,E2 22182.38} C_VEL
LIN {X 0,Y 496.77,Z 612.354,A -85,B 0,C 180,E1 22178.837,E2 22178.837} C_VEL
LIN {X 0,Y 496.763,Z 612.355,A -85,B 0,C 180,E1 22175.196,E2 22175.196} C_VEL
LIN {X 0,Y 496.758,Z 612.353,A -85,B 0,C 180,E1 22171.635,E2 22171.635} C_VEL
LIN {X 0,Y 496.748,Z 612.357,A -85,B 0,C 180,E1 22168.099,E2 22168.099} C_VEL
LIN {X 0,Y 496.769,Z 612.358,A -85,B 0,C 180,E1 22164.528,E2 22164.528} C_VEL
LIN {X 0,Y 496.769,Z 612.354,A -85,B 0,C 180,E1 22160.947,E2 22160.947} C_VEL
LIN {X 0,Y 496.732,Z 612.359,A -85,B 0,C 180,E1 22157.425,E2 22157.425} C_VEL
LIN {X 0,Y 496.744,Z 612.361,A -85,B 0,C 180,E1 22153.858,E2 22153.858} C_VEL
LIN {X 0,Y 496.765,Z 612.357,A -85,B 0,C 180,E1 22150.436,E2 22150.436} C_VEL
LIN {X 0,Y 496.764,Z 612.579,A -85,B 0,C 180,E1 22147.619,E2 22147.619} C_VEL
LIN {X 0,Y 500.742,Z 628.249,A -85,B 0,C 180,E1 22145.672,E2 22145.672} C_VEL
LIN {X 0,Y 500.914,Z 650.012,A -85,B 0,C 180,E1 22143.261,E2 22143.261} C_VEL
LIN {X 0,Y 500.676,Z 678.705,A -85,B 0,C 180,E1 22140,E2 22140} C_VEL
LIN {X 0,Y 500.383,Z 703.316,A -85,B 0,C 180,E1 22137.17,E2 22137.17} C_VEL
LIN {X 0,Y 501.007,Z 707.996,A -85,B 0,C 180,E1 22137.061,E2 22137.061} C_VEL
LIN {X 0,Y 499.863,Z 842.49,A -85,B 0,C 180,E1 22134.982,E2 22134.982} C_VEL
LIN {X 0,Y 499.72,Z 858.279,A -85,B 0,C 180,E1 22134.526,E2 22134.526} C_VEL
LIN {X 0,Y 499.432,Z 873.995,A -85,B 0,C 180,E1 22133.851,E2 22133.851} C_VEL
LIN {X 0,Y 499.065,Z 887.948,A -85,B 0,C 180,E1 22133.038,E2 22133.038} C_VEL
LIN {X 0,Y 498.582,Z 902.539,A -85,B 0,C 180,E1 22131.93,E2 22131.93} C_VEL
LIN {X 0,Y 498.118,Z 914.664,A -85,B 0,C 180,E1 22130.759,E2 22130.759} C_VEL
LIN {X 0,Y 497.632,Z 926.344,A -85,B 0,C 180,E1 22129.347,E2 22129.347} C_VEL
LIN {X 0,Y 497.236,Z 935.738,A -85,B 0,C 180,E1 22127.929,E2 22127.929} C_VEL
LIN {X 0,Y 496.893,Z 944.422,A -85,B 0,C 180,E1 22126.264,E2 22126.264} C_VEL
LIN {X 0,Y 496.659,Z 951.154,A -85,B 0,C 180,E1 22124.589,E2 22124.589} C_VEL
LIN {X 0,Y 496.473,Z 956.697,A -85,B 0,C 180,E1 22122.67,E2 22122.67} C_VEL
LIN {X 0,Y 496.371,Z 960.121,A -85,B 0,C 180,E1 22120.832,E2 22120.832} C_VEL
LIN {X 0,Y 496.323,Z 961.876,A -85,B 0,C 180,E1 22118.863,E2 22118.863} C_VEL
LIN {X 0,Y 496.315,Z 961.77,A -85,B 0,C 180,E1 22116.994,E2 22116.994} C_VEL
LIN {X 0,Y 496.341,Z 959.735,A -85,B 0,C 180,E1 22114.973,E2 22114.973} C_VEL
LIN {X 0,Y 496.417,Z 956.116,A -85,B 0,C 180,E1 22113.161,E2 22113.161} C_VEL
LIN {X 0,Y 496.565,Z 950.769,A -85,B 0,C 180,E1 22111.365,E2 22111.365} C_VEL
LIN {X 0,Y 496.786,Z 943.813,A -85,B 0,C 180,E1 22109.657,E2 22109.657} C_VEL
LIN {X 0,Y 497.125,Z 934.629,A -85,B 0,C 180,E1 22107.928,E2 22107.928} C_VEL
LIN {X 0,Y 497.253,Z 931.316,A -85,B 0,C 180,E1 22107.404,E2 22107.404} C_VEL
LIN {X 0,Y 496.485,Z 926.703,A -85,B 0,C 180,E1 22106.689,E2 22106.689} C_VEL
LIN {X 0,Y 491.94,Z 916.569,A -85,B 0,C 180,E1 22105.234,E2 22105.234} C_VEL
LIN {X 0,Y 490.553,Z 911.198,A -85,B 0,C 180,E1 22104.598,E2 22104.598} C_VEL
LIN {X 0,Y 490.471,Z 908.678,A -85,B 0,C 180,E1 22104.338,E2 22104.338} C_VEL
LIN {X 0,Y 490.955,Z 895.776,A -85,B 0,C 180,E1 22103.219,E2 22103.219} C_VEL
LIN {X 0,Y 491.439,Z 881.412,A -85,B 0,C 180,E1 22102.236,E2 22102.236} C_VEL
LIN {X 0,Y 491.844,Z 866.365,A -85,B 0,C 180,E1 22101.458,E2 22101.458} C_VEL
LIN {X 0,Y 492.134,Z 849.683,A -85,B 0,C 180,E1 22100.846,E2 22100.846} C_VEL
LIN {X 0,Y 492.25,Z 832.811,A -85,B 0,C 180,E1 22100.471,E2 22100.471} C_VEL
LIN {X 0,Y 493.185,Z 706.268,A -85,B 0,C 180,E1 22098.524,E2 22098.524} C_VEL
LIN {X 0,Y 492.086,Z 700.491,A -85,B 0,C 180,E1 22098.361,E2 22098.361} C_VEL
LIN {X 0,Y 492.704,Z 671.579,A -85,B 0,C 180,E1 22094.908,E2 22094.908} C_VEL
LIN {X 0,Y 493.272,Z 641.001,A -85,B 0,C 180,E1 22091.276,E2 22091.276} C_VEL
LIN {X 0,Y 493.189,Z 630.875,A -85,B 0,C 180,E1 22090.067,E2 22090.067} C_VEL
LIN {X 0,Y 488.85,Z 613.5,A -85,B 0,C 180,E1 22087.726,E2 22087.726} C_VEL
LIN {X 0,Y 488.78,Z 613.35,A -85,B 0,C 180,E1 22084.232,E2 22084.232} C_VEL
LIN {X 0,Y 488.773,Z 613.347,A -85,B 0,C 180,E1 22080.758,E2 22080.758} C_VEL
LIN {X 0,Y 488.834,Z 613.345,A -85,B 0,C 180,E1 22077.401,E2 22077.401} C_VEL
LIN {X 0,Y 488.782,Z 613.329,A -85,B 0,C 180,E1 22073.88,E2 22073.88} C_VEL
LIN {X 0,Y 488.782,Z 613.335,A -85,B 0,C 180,E1 22070.35,E2 22070.35} C_VEL
LIN {X 0,Y 488.831,Z 613.334,A -85,B 0,C 180,E1 22066.885,E2 22066.885} C_VEL
LIN {X 0,Y 488.842,Z 613.618,A -85,B 0,C 180,E1 22064.375,E2 22064.375} C_VEL
LIN {X 0,Y 494.118,Z 632.731,A -85,B 0,C 180,E1 22061.32,E2 22061.32} C_VEL
LIN {X 0,Y 494.64,Z 636.486,A -85,B 0,C 180,E1 22060.766,E2 22060.766} C_VEL
LIN {X 0,Y 493.283,Z 664.038,A -85,B 0,C 180,E1 22057.103,E2 22057.103} C_VEL
LIN {X 0,Y 491.973,Z 693.358,A -85,B 0,C 180,E1 22053.263,E2 22053.263} C_VEL
LIN {X 0,Y 492.824,Z 697.962,A -85,B 0,C 180,E1 22053.093,E2 22053.093} C_VEL
LIN {X 0,Y 494.994,Z 709.272,A -85,B 0,C 180,E1 22052.813,E2 22052.813} C_VEL
LIN {X 0,Y 493.736,Z 838.304,A -85,B 0,C 180,E1 22050.845,E2 22050.845} C_VEL
LIN {X 0,Y 493.412,Z 855.237,A -85,B 0,C 180,E1 22050.356,E2 22050.356} C_VEL
LIN {X 0,Y 492.941,Z 870.976,A -85,B 0,C 180,E1 22049.678,E2 22049.678} C_VEL
LIN {X 0,Y 492.314,Z 886.22,A -85,B 0,C 180,E1 22048.778,E2 22048.778} C_VEL
LIN {X 0,Y 491.644,Z 900.073,A -85,B 0,C 180,E1 22047.728,E2 22047.728} C_VEL
LIN {X 0,Y 490.959,Z 912.857,A -85,B 0,C 180,E1 22046.498,E2 22046.498} C_VEL
LIN {X 0,Y 490.291,Z 924.649,A -85,B 0,C 180,E1 22045.087,E2 22045.087} C_VEL
LIN {X 0,Y 489.7,Z 934.934,A -85,B 0,C 180,E1 22043.553,E2 22043.553} C_VEL
LIN {X 0,Y 489.187,Z 944.295,A -85,B 0,C 180,E1 22041.775,E2 22041.775} C_VEL
LIN {X 0,Y 488.846,Z 951.519,A -85,B 0,C 180,E1 22039.988,E2 22039.988} C_VEL
LIN {X 0,Y 488.618,Z 957.165,A -85,B 0,C 180,E1 22038.073,E2 22038.073} C_VEL
LIN {X 0,Y 488.483,Z 960.979,A -85,B 0,C 180,E1 22036.144,E2 22036.144} C_VEL
LIN {X 0,Y 488.42,Z 962.975,A -85,B 0,C 180,E1 22034.187,E2 22034.187} C_VEL
LIN {X 0,Y 488.423,Z 963.257,A -85,B 0,C 180,E1 22032.16,E2 22032.16} C_VEL
LIN {X 0,Y 488.483,Z 961.602,A -85,B 0,C 180,E1 22030.137,E2 22030.137} C_VEL
LIN {X 0,Y 488.616,Z 958.393,A -85,B 0,C 180,E1 22028.261,E2 22028.261} C_VEL
LIN {X 0,Y 488.831,Z 953.423,A -85,B 0,C 180,E1 22026.398,E2 22026.398} C_VEL
LIN {X 0,Y 489.159,Z 946.699,A -85,B 0,C 180,E1 22024.58,E2 22024.58} C_VEL
LIN {X 0,Y 489.62,Z 938.66,A -85,B 0,C 180,E1 22022.91,E2 22022.91} C_VEL
LIN {X 0,Y 490.214,Z 928.669,A -85,B 0,C 180,E1 22021.289,E2 22021.289} C_VEL
LIN {X 0,Y 490.918,Z 917.196,A -85,B 0,C 180,E1 22019.797,E2 22019.797} C_VEL
LIN {X 0,Y 491.629,Z 904.505,A -85,B 0,C 180,E1 22018.488,E2 22018.488} C_VEL
LIN {X 0,Y 492.345,Z 890.809,A -85,B 0,C 180,E1 22017.361,E2 22017.361} C_VEL
LIN {X 0,Y 492.992,Z 876.244,A -85,B 0,C 180,E1 22016.428,E2 22016.428} C_VEL
LIN {X 0,Y 493.561,Z 860.082,A -85,B 0,C 180,E1 22015.654,E2 22015.654} C_VEL
LIN {X 0,Y 493.927,Z 844.138,A -85,B 0,C 180,E1 22015.124,E2 22015.124} C_VEL
LIN {X 0,Y 494.144,Z 824.839,A -85,B 0,C 180,E1 22014.752,E2 22014.752} C_VEL
LIN {X 0,Y 495.227,Z 707.578,A -85,B 0,C 180,E1 22012.953,E2 22012.953} C_VEL
LIN {X 0,Y 492.36,Z 694.301,A -85,B 0,C 180,E1 22012.564,E2 22012.564} C_VEL
LIN {X 0,Y 492.399,Z 690.497,A -85,B 0,C 180,E1 22012.124,E2 22012.124} C_VEL
LIN {X 0,Y 493.821,Z 662.461,A -85,B 0,C 180,E1 22008.386,E2 22008.386} C_VEL
LIN {X 0,Y 495.297,Z 636.324,A -85,B 0,C 180,E1 22004.839,E2 22004.839} C_VEL
LIN {X 0,Y 490.974,Z 620.573,A -85,B 0,C 180,E1 22002.225,E2 22002.225} C_VEL
LIN {X 0,Y 488.84,Z 613.434,A -85,B 0,C 180,E1 22000.921,E2 22000.921} C_VEL
LIN {X 0,Y 488.818,Z 613.346,A -85,B 0,C 180,E1 21997.262,E2 21997.262} C_VEL
LIN {X 0,Y 488.826,Z 613.34,A -85,B 0,C 180,E1 21993.645,E2 21993.645} C_VEL
LIN {X 0,Y 488.822,Z 613.347,A -85,B 0,C 180,E1 21990.075,E2 21990.075} C_VEL
LIN {X 0,Y 488.824,Z 613.346,A -85,B 0,C 180,E1 21986.482,E2 21986.482} C_VEL
LIN {X 0,Y 488.827,Z 613.34,A -85,B 0,C 180,E1 21982.87,E2 21982.87} C_VEL
LIN {X 0,Y 488.814,Z 613.339,A -85,B 0,C 180,E1 21979.352,E2 21979.352} C_VEL
LIN {X 0,Y 488.829,Z 613.344,A -85,B 0,C 180,E1 21975.786,E2 21975.786} C_VEL
LIN {X 0,Y 488.822,Z 613.344,A -85,B 0,C 180,E1 21972.163,E2 21972.163} C_VEL
LIN {X 0,Y 488.821,Z 613.341,A -85,B 0,C 180,E1 21968.588,E2 21968.588} C_VEL
LIN {X 0,Y 488.812,Z 613.34,A -85,B 0,C 180,E1 21964.929,E2 21964.929} C_VEL
LIN {X 0,Y 488.825,Z 613.339,A -85,B 0,C 180,E1 21961.407,E2 21961.407} C_VEL
LIN {X 0,Y 488.828,Z 613.341,A -85,B 0,C 180,E1 21957.773,E2 21957.773} C_VEL
LIN {X 0,Y 488.809,Z 613.342,A -85,B 0,C 180,E1 21954.248,E2 21954.248} C_VEL
LIN {X 0,Y 488.823,Z 613.334,A -85,B 0,C 180,E1 21950.701,E2 21950.701} C_VEL
LIN {X 0,Y 488.826,Z 613.341,A -85,B 0,C 180,E1 21947.118,E2 21947.118} C_VEL
LIN {X 0,Y 488.814,Z 613.343,A -85,B 0,C 180,E1 21943.603,E2 21943.603} C_VEL
LIN {X 0,Y 488.814,Z 613.346,A -85,B 0,C 180,E1 21940.026,E2 21940.026} C_VEL
LIN {X 0,Y 488.826,Z 613.335,A -85,B 0,C 180,E1 21936.493,E2 21936.493} C_VEL
LIN {X 0,Y 488.818,Z 613.336,A -85,B 0,C 180,E1 21932.994,E2 21932.994} C_VEL
LIN {X 0,Y 488.804,Z 613.338,A -85,B 0,C 180,E1 21929.381,E2 21929.381} C_VEL
LIN {X 0,Y 488.828,Z 613.343,A -85,B 0,C 180,E1 21925.914,E2 21925.914} C_VEL
LIN {X 0,Y 488.83,Z 613.34,A -85,B 0,C 180,E1 21922.296,E2 21922.296} C_VEL
LIN {X 0,Y 488.801,Z 613.343,A -85,B 0,C 180,E1 21918.802,E2 21918.802} C_VEL
LIN {X 0,Y 488.822,Z 613.349,A -85,B 0,C 180,E1 21915.216,E2 21915.216} C_VEL
LIN {X 0,Y 488.831,Z 613.341,A -85,B 0,C 180,E1 21911.663,E2 21911.663} C_VEL
LIN {X 0,Y 488.802,Z 613.346,A -85,B 0,C 180,E1 21908.152,E2 21908.152} C_VEL
LIN {X 0,Y 488.898,Z 613.779,A -85,B 0,C 180,E1 21907.594,E2 21907.594} C_VEL
LIN {X 0,Y 495.879,Z 633.392,A -85,B 0,C 180,E1 21905.152,E2 21905.152} C_VEL
LIN {X 0,Y 499.112,Z 643.056,A -85,B 0,C 180,E1 21904.05,E2 21904.05} C_VEL
LIN {X 0,Y 496.855,Z 687.18,A -85,B 0,C 180,E1 21900.338,E2 21900.338} C_VEL
LIN {X 0,Y 495.989,Z 709.021,A -85,B 0,C 180,E1 21898.573,E2 21898.573} C_VEL
LIN {X 0,Y 498.605,Z 727.988,A -85,B 0,C 180,E1 21898.137,E2 21898.137} C_VEL
LIN {X 0,Y 496.615,Z 926.139,A -85,B 0,C 180,E1 21895.183,E2 21895.183} C_VEL
LIN {X 0,Y 496.013,Z 945.768,A -85,B 0,C 180,E1 21894.678,E2 21894.678} C_VEL
LIN {X 0,Y 495.268,Z 964.692,A -85,B 0,C 180,E1 21893.972,E2 21893.972} C_VEL
LIN {X 0,Y 494.423,Z 982.45,A -85,B 0,C 180,E1 21893.099,E2 21893.099} C_VEL
LIN {X 0,Y 493.464,Z 999.978,A -85,B 0,C 180,E1 21892.015,E2 21892.015} C_VEL
LIN {X 0,Y 492.473,Z 1016.657,A -85,B 0,C 180,E1 21890.749,E2 21890.749} C_VEL
LIN {X 0,Y 491.493,Z 1032.64,A -85,B 0,C 180,E1 21889.278,E2 21889.278} C_VEL
LIN {X 0,Y 490.634,Z 1045.748,A -85,B 0,C 180,E1 21887.799,E2 21887.799} C_VEL
LIN {X 0,Y 489.765,Z 1058.986,A -85,B 0,C 180,E1 21885.998,E2 21885.998} C_VEL
LIN {X 0,Y 489.077,Z 1070.665,A -85,B 0,C 180,E1 21884.08,E2 21884.08} C_VEL
LIN {X 0,Y 488.569,Z 1080.824,A -85,B 0,C 180,E1 21882.048,E2 21882.048} C_VEL
LIN {X 0,Y 488.228,Z 1089.434,A -85,B 0,C 180,E1 21879.905,E2 21879.905} C_VEL
LIN {X 0,Y 488.033,Z 1096.129,A -85,B 0,C 180,E1 21877.771,E2 21877.771} C_VEL
LIN {X 0,Y 487.942,Z 1101.294,A -85,B 0,C 180,E1 21875.526,E2 21875.526} C_VEL
LIN {X 0,Y 487.914,Z 1104.656,A -85,B 0,C 180,E1 21873.289,E2 21873.289} C_VEL
LIN {X 0,Y 487.907,Z 1106.303,A -85,B 0,C 180,E1 21871.056,E2 21871.056} C_VEL
LIN {X 0,Y 487.906,Z 1106.266,A -85,B 0,C 180,E1 21868.825,E2 21868.825} C_VEL
LIN {X 0,Y 487.914,Z 1104.539,A -85,B 0,C 180,E1 21866.593,E2 21866.593} C_VEL
LIN {X 0,Y 487.946,Z 1101.084,A -85,B 0,C 180,E1 21864.355,E2 21864.355} C_VEL
LIN {X 0,Y 488.042,Z 1095.817,A -85,B 0,C 180,E1 21862.11,E2 21862.11} C_VEL
LIN {X 0,Y 488.24,Z 1089.024,A -85,B 0,C 180,E1 21859.975,E2 21859.975} C_VEL
LIN {X 0,Y 488.594,Z 1080.297,A -85,B 0,C 180,E1 21857.832,E2 21857.832} C_VEL
LIN {X 0,Y 489.117,Z 1070.002,A -85,B 0,C 180,E1 21855.8,E2 21855.8} C_VEL
LIN {X 0,Y 489.818,Z 1058.163,A -85,B 0,C 180,E1 21853.882,E2 21853.882} C_VEL
LIN {X 0,Y 490.695,Z 1044.738,A -85,B 0,C 180,E1 21852.08,E2 21852.08} C_VEL
LIN {X 0,Y 491.551,Z 1031.827,A -85,B 0,C 180,E1 21850.636,E2 21850.636} C_VEL
LIN {X 0,Y 492.55,Z 1015.557,A -85,B 0,C 180,E1 21849.155,E2 21849.155} C_VEL
LIN {X 0,Y 493.568,Z 998.283,A -85,B 0,C 180,E1 21847.864,E2 21847.864} C_VEL
LIN {X 0,Y 494.539,Z 980.36,A -85,B 0,C 180,E1 21846.78,E2 21846.78} C_VEL
LIN {X 0,Y 495.409,Z 962.047,A -85,B 0,C 180,E1 21845.908,E2 21845.908} C_VEL
LIN {X 0,Y 496.136,Z 942.948,A -85,B 0,C 180,E1 21845.229,E2 21845.229} C_VEL
LIN {X 0,Y 496.682,Z 923.567,A -85,B 0,C 180,E1 21844.761,E2 21844.761} C_VEL
LIN {X 0,Y 498.502,Z 725.502,A -85,B 0,C 180,E1 21841.804,E2 21841.804} C_VEL
LIN {X 0,Y 496.026,Z 708.566,A -85,B 0,C 180,E1 21841.384,E2 21841.384} C_VEL
LIN {X 0,Y 497.877,Z 666.663,A -85,B 0,C 180,E1 21837.938,E2 21837.938} C_VEL
LIN {X 0,Y 499.115,Z 642.53,A -85,B 0,C 180,E1 21835.881,E2 21835.881} C_VEL
LIN {X 0,Y 490.719,Z 618.927,A -85,B 0,C 180,E1 21833.104,E2 21833.104} C_VEL
LIN {X 0,Y 488.86,Z 613.549,A -85,B 0,C 180,E1 21832.397,E2 21832.397} C_VEL
LIN {X 0,Y 488.829,Z 613.347,A -85,B 0,C 180,E1 21828.804,E2 21828.804} C_VEL
LIN {X 0,Y 488.819,Z 613.345,A -85,B 0,C 180,E1 21825.216,E2 21825.216} C_VEL
LIN {X 0,Y 488.82,Z 613.342,A -85,B 0,C 180,E1 21821.527,E2 21821.527} C_VEL
LIN {X 0,Y 488.818,Z 613.343,A -85,B 0,C 180,E1 21818.002,E2 21818.002} C_VEL
LIN {X 0,Y 488.82,Z 613.348,A -85,B 0,C 180,E1 21814.371,E2 21814.371} C_VEL
LIN {X 0,Y 488.829,Z 613.345,A -85,B 0,C 180,E1 21810.754,E2 21810.754} C_VEL
LIN {X 0,Y 488.831,Z 613.341,A -85,B 0,C 180,E1 21807.137,E2 21807.137} C_VEL
LIN {X 0,Y 488.801,Z 613.345,A -85,B 0,C 180,E1 21803.594,E2 21803.594} C_VEL
LIN {X 0,Y 488.807,Z 613.349,A -85,B 0,C 180,E1 21799.974,E2 21799.974} C_VEL
LIN {X 0,Y 488.833,Z 613.346,A -85,B 0,C 180,E1 21796.395,E2 21796.395} C_VEL
LIN {X 0,Y 488.802,Z 613.347,A -85,B 0,C 180,E1 21792.883,E2 21792.883} C_VEL
LIN {X 0,Y 488.782,Z 613.351,A -85,B 0,C 180,E1 21789.3,E2 21789.3} C_VEL
LIN {X 0,Y 488.866,Z 613.592,A -85,B 0,C 180,E1 21787.994,E2 21787.994} C_VEL
LIN {X 0,Y 493.112,Z 630.018,A -85,B 0,C 180,E1 21785.935,E2 21785.935} C_VEL
LIN {X 0,Y 493.456,Z 635.266,A -85,B 0,C 180,E1 21785.348,E2 21785.348} C_VEL
LIN {X 0,Y 493.349,Z 662.266,A -85,B 0,C 180,E1 21782.323,E2 21782.323} C_VEL
LIN {X 0,Y 493.052,Z 688.673,A -85,B 0,C 180,E1 21779.303,E2 21779.303} C_VEL
LIN {X 0,Y 492.863,Z 704.547,A -85,B 0,C 180,E1 21777.471,E2 21777.471} C_VEL
LIN {X 0,Y 493.472,Z 709.158,A -85,B 0,C 180,E1 21777.358,E2 21777.358} C_VEL
LIN {X 0,Y 492.208,Z 843.964,A -85,B 0,C 180,E1 21775.225,E2 21775.225} C_VEL
LIN {X 0,Y 492.063,Z 859.919,A -85,B 0,C 180,E1 21774.753,E2 21774.753} C_VEL
LIN {X 0,Y 491.76,Z 875.963,A -85,B 0,C 180,E1 21774.048,E2 21774.048} C_VEL
LIN {X 0,Y 491.343,Z 890.587,A -85,B 0,C 180,E1 21773.163,E2 21773.163} C_VEL
LIN {X 0,Y 490.869,Z 904.248,A -85,B 0,C 180,E1 21772.097,E2 21772.097} C_VEL
LIN {X 0,Y 490.347,Z 916.819,A -85,B 0,C 180,E1 21770.848,E2 21770.848} C_VEL
LIN {X 0,Y 489.835,Z 928.364,A -85,B 0,C 180,E1 21769.414,E2 21769.414} C_VEL
LIN {X 0,Y 489.376,Z 938.266,A -85,B 0,C 180,E1 21767.851,E2 21767.851} C_VEL
LIN {X 0,Y 489.024,Z 946.714,A -85,B 0,C 180,E1 21766.159,E2 21766.159} C_VEL
LIN {X 0,Y 488.75,Z 953.548,A -85,B 0,C 180,E1 21764.333,E2 21764.333} C_VEL
LIN {X 0,Y 488.572,Z 958.511,A -85,B 0,C 180,E1 21762.492,E2 21762.492} C_VEL
LIN {X 0,Y 488.461,Z 961.803,A -85,B 0,C 180,E1 21760.509,E2 21760.509} C_VEL
LIN {X 0,Y 488.415,Z 963.181,A -85,B 0,C 180,E1 21758.629,E2 21758.629} C_VEL
LIN {X 0,Y 488.404,Z 962.734,A -85,B 0,C 180,E1 21756.599,E2 21756.599} C_VEL
LIN {X 0,Y 488.444,Z 960.713,A -85,B 0,C 180,E1 21754.796,E2 21754.796} C_VEL
LIN {X 0,Y 488.538,Z 956.66,A -85,B 0,C 180,E1 21752.845,E2 21752.845} C_VEL
LIN {X 0,Y 488.709,Z 951.42,A -85,B 0,C 180,E1 21751.123,E2 21751.123} C_VEL
LIN {X 0,Y 488.954,Z 944.26,A -85,B 0,C 180,E1 21749.391,E2 21749.391} C_VEL
LIN {X 0,Y 489.324,Z 935.267,A -85,B 0,C 180,E1 21747.701,E2 21747.701} C_VEL
LIN {X 0,Y 489.781,Z 924.54,A -85,B 0,C 180,E1 21746.129,E2 21746.129} C_VEL
LIN {X 0,Y 490.297,Z 912.786,A -85,B 0,C 180,E1 21744.751,E2 21744.751} C_VEL
LIN {X 0,Y 490.471,Z 908.678,A -85,B 0,C 180,E1 21744.338,E2 21744.338} C_VEL
LIN {X 0,Y 489.771,Z 902.821,A -85,B 0,C 180,E1 21743.744,E2 21743.744} C_VEL
LIN {X 0,Y 485.898,Z 891.923,A -85,B 0,C 180,E1 21742.706,E2 21742.706} C_VEL
LIN {X 0,Y 484.031,Z 884.631,A -85,B 0,C 180,E1 21742.144,E2 21742.144} C_VEL
LIN {X 0,Y 483.81,Z 880.709,A -85,B 0,C 180,E1 21741.901,E2 21741.901} C_VEL
LIN {X 0,Y 484.225,Z 865.155,A -85,B 0,C 180,E1 21741.118,E2 21741.118} C_VEL
LIN {X 0,Y 484.492,Z 849.333,A -85,B 0,C 180,E1 21740.554,E2 21740.554} C_VEL
LIN {X 0,Y 484.598,Z 831.369,A -85,B 0,C 180,E1 21740.174,E2 21740.174} C_VEL
LIN {X 0,Y 485.635,Z 707.434,A -85,B 0,C 180,E1 21738.229,E2 21738.229} C_VEL
LIN {X 0,Y 484.505,Z 701.267,A -85,B 0,C 180,E1 21738.038,E2 21738.038} C_VEL
LIN {X 0,Y 485.146,Z 671.608,A -85,B 0,C 180,E1 21734.485,E2 21734.485} C_VEL
LIN {X 0,Y 485.707,Z 642.724,A -85,B 0,C 180,E1 21731.048,E2 21731.048} C_VEL
LIN {X 0,Y 485.604,Z 633.093,A -85,B 0,C 180,E1 21729.895,E2 21729.895} C_VEL
LIN {X 0,Y 480.875,Z 614.497,A -85,B 0,C 180,E1 21727.363,E2 21727.363} C_VEL
LIN {X 0,Y 480.864,Z 614.331,A -85,B 0,C 180,E1 21723.938,E2 21723.938} C_VEL
LIN {X 0,Y 480.831,Z 614.336,A -85,B 0,C 180,E1 21720.49,E2 21720.49} C_VEL
LIN {X 0,Y 480.873,Z 614.332,A -85,B 0,C 180,E1 21717.088,E2 21717.088} C_VEL
LIN {X 0,Y 480.872,Z 614.318,A -85,B 0,C 180,E1 21713.514,E2 21713.514} C_VEL
LIN {X 0,Y 480.837,Z 614.321,A -85,B 0,C 180,E1 21710.066,E2 21710.066} C_VEL
LIN {X 0,Y 480.868,Z 614.32,A -85,B 0,C 180,E1 21706.551,E2 21706.551} C_VEL
LIN {X 0,Y 480.931,Z 614.565,A -85,B 0,C 180,E1 21704.834,E2 21704.834} C_VEL
LIN {X 0,Y 486.359,Z 634.317,A -85,B 0,C 180,E1 21701.623,E2 21701.623} C_VEL
LIN {X 0,Y 487.144,Z 638.385,A -85,B 0,C 180,E1 21701.005,E2 21701.005} C_VEL
LIN {X 0,Y 485.698,Z 665.655,A -85,B 0,C 180,E1 21697.333,E2 21697.333} C_VEL
LIN {X 0,Y 484.376,Z 693.629,A -85,B 0,C 180,E1 21693.64,E2 21693.64} C_VEL
LIN {X 0,Y 486.18,Z 702.473,A -85,B 0,C 180,E1 21693.367,E2 21693.367} C_VEL
LIN {X 0,Y 487.64,Z 710.594,A -85,B 0,C 180,E1 21693.167,E2 21693.167} C_VEL
LIN {X 0,Y 486.29,Z 838.998,A -85,B 0,C 180,E1 21691.178,E2 21691.178} C_VEL
LIN {X 0,Y 485.948,Z 855.963,A -85,B 0,C 180,E1 21690.682,E2 21690.682} C_VEL
LIN {X 0,Y 485.455,Z 871.637,A -85,B 0,C 180,E1 21690,E2 21690} C_VEL
LIN {X 0,Y 484.803,Z 886.549,A -85,B 0,C 180,E1 21689.114,E2 21689.114} C_VEL
LIN {X 0,Y 484.079,Z 900.532,A -85,B 0,C 180,E1 21688.047,E2 21688.047} C_VEL
LIN {X 0,Y 483.343,Z 913.446,A -85,B 0,C 180,E1 21686.798,E2 21686.798} C_VEL
LIN {X 0,Y 482.61,Z 925.318,A -85,B 0,C 180,E1 21685.366,E2 21685.366} C_VEL
LIN {X 0,Y 481.962,Z 935.701,A -85,B 0,C 180,E1 21683.807,E2 21683.807} C_VEL
LIN {X 0,Y 481.42,Z 944.566,A -85,B 0,C 180,E1 21682.122,E2 21682.122} C_VEL
LIN {X 0,Y 481.027,Z 952.011,A -85,B 0,C 180,E1 21680.307,E2 21680.307} C_VEL
LIN {X 0,Y 480.756,Z 957.752,A -85,B 0,C 180,E1 21678.4,E2 21678.4} C_VEL
LIN {X 0,Y 480.594,Z 961.837,A -85,B 0,C 180,E1 21676.403,E2 21676.403} C_VEL
LIN {X 0,Y 480.514,Z 964.033,A -85,B 0,C 180,E1 21674.43,E2 21674.43} C_VEL
LIN {X 0,Y 480.51,Z 964.48,A -85,B 0,C 180,E1 21672.314,E2 21672.314} C_VEL
LIN {X 0,Y 480.57,Z 963.239,A -85,B 0,C 180,E1 21670.429,E2 21670.429} C_VEL
LIN {X 0,Y 480.712,Z 960.05,A -85,B 0,C 180,E1 21668.395,E2 21668.395} C_VEL
LIN {X 0,Y 480.957,Z 955.236,A -85,B 0,C 180,E1 21666.463,E2 21666.463} C_VEL
LIN {X 0,Y 481.298,Z 948.835,A -85,B 0,C 180,E1 21664.647,E2 21664.647} C_VEL
LIN {X 0,Y 481.822,Z 940.47,A -85,B 0,C 180,E1 21662.836,E2 21662.836} C_VEL
LIN {X 0,Y 482.444,Z 931.058,A -85,B 0,C 180,E1 21661.243,E2 21661.243} C_VEL
LIN {X 0,Y 483.215,Z 919.448,A -85,B 0,C 180,E1 21659.677,E2 21659.677} C_VEL
LIN {X 0,Y 484.001,Z 906.999,A -85,B 0,C 180,E1 21658.334,E2 21658.334} C_VEL
LIN {X 0,Y 484.789,Z 893.136,A -85,B 0,C 180,E1 21657.151,E2 21657.151} C_VEL
LIN {X 0,Y 485.476,Z 879.242,A -85,B 0,C 180,E1 21656.215,E2 21656.215} C_VEL
LIN {X 0,Y 486.073,Z 864.137,A -85,B 0,C 180,E1 21655.444,E2 21655.444} C_VEL
LIN {X 0,Y 486.519,Z 847.318,A -85,B 0,C 180,E1 21654.836,E2 21654.836} C_VEL
LIN {X 0,Y 486.745,Z 830.652,A -85,B 0,C 180,E1 21654.47,E2 21654.47} C_VEL
LIN {X 0,Y 487.997,Z 708.899,A -85,B 0,C 180,E1 21652.569,E2 21652.569} C_VEL
LIN {X 0,Y 484.814,Z 694.199,A -85,B 0,C 180,E1 21652.123,E2 21652.123} C_VEL
LIN {X 0,Y 486.248,Z 666.153,A -85,B 0,C 180,E1 21648.381,E2 21648.381} C_VEL
LIN {X 0,Y 487.911,Z 639.093,A -85,B 0,C 180,E1 21644.66,E2 21644.66} C_VEL
LIN {X 0,Y 483.691,Z 623.65,A -85,B 0,C 180,E1 21642.049,E2 21642.049} C_VEL
LIN {X 0,Y 480.895,Z 614.441,A -85,B 0,C 180,E1 21640.351,E2 21640.351} C_VEL
LIN {X 0,Y 480.887,Z 614.335,A -85,B 0,C 180,E1 21636.785,E2 21636.785} C_VEL
LIN {X 0,Y 480.882,Z 614.331,A -85,B 0,C 180,E1 21633.15,E2 21633.15} C_VEL
LIN {X 0,Y 480.885,Z 614.331,A -85,B 0,C 180,E1 21629.523,E2 21629.523} C_VEL
LIN {X 0,Y 480.881,Z 614.328,A -85,B 0,C 180,E1 21625.89,E2 21625.89} C_VEL
LIN {X 0,Y 480.887,Z 614.327,A -85,B 0,C 180,E1 21622.236,E2 21622.236} C_VEL
LIN {X 0,Y 480.883,Z 614.325,A -85,B 0,C 180,E1 21618.537,E2 21618.537} C_VEL
LIN {X 0,Y 480.878,Z 614.324,A -85,B 0,C 180,E1 21614.941,E2 21614.941} C_VEL
LIN {X 0,Y 480.877,Z 614.329,A -85,B 0,C 180,E1 21611.271,E2 21611.271} C_VEL
LIN {X 0,Y 480.889,Z 614.335,A -85,B 0,C 180,E1 21607.647,E2 21607.647} C_VEL
LIN {X 0,Y 480.885,Z 614.328,A -85,B 0,C 180,E1 21603.935,E2 21603.935} C_VEL
LIN {X 0,Y 480.874,Z 614.323,A -85,B 0,C 180,E1 21600.358,E2 21600.358} C_VEL
LIN {X 0,Y 480.873,Z 614.324,A -85,B 0,C 180,E1 21596.663,E2 21596.663} C_VEL
LIN {X 0,Y 480.889,Z 614.333,A -85,B 0,C 180,E1 21593.074,E2 21593.074} C_VEL
LIN {X 0,Y 480.887,Z 614.325,A -85,B 0,C 180,E1 21589.457,E2 21589.457} C_VEL
LIN {X 0,Y 480.869,Z 614.323,A -85,B 0,C 180,E1 21585.92,E2 21585.92} C_VEL
LIN {X 0,Y 480.884,Z 614.327,A -85,B 0,C 180,E1 21582.328,E2 21582.328} C_VEL
LIN {X 0,Y 480.887,Z 614.334,A -85,B 0,C 180,E1 21578.663,E2 21578.663} C_VEL
LIN {X 0,Y 480.882,Z 614.331,A -85,B 0,C 180,E1 21575.031,E2 21575.031} C_VEL
LIN {X 0,Y 480.867,Z 614.335,A -85,B 0,C 180,E1 21571.43,E2 21571.43} C_VEL
LIN {X 0,Y 480.889,Z 614.329,A -85,B 0,C 180,E1 21567.841,E2 21567.841} C_VEL
LIN {X 0,Y 480.889,Z 614.329,A -85,B 0,C 180,E1 21564.182,E2 21564.182} C_VEL
LIN {X 0,Y 480.868,Z 614.335,A -85,B 0,C 180,E1 21560.641,E2 21560.641} C_VEL
LIN {X 0,Y 480.869,Z 614.332,A -85,B 0,C 180,E1 21557,E2 21557} C_VEL
LIN {X 0,Y 480.891,Z 614.33,A -85,B 0,C 180,E1 21553.479,E2 21553.479} C_VEL
LIN {X 0,Y 480.888,Z 614.33,A -85,B 0,C 180,E1 21549.821,E2 21549.821} C_VEL
LIN {X 0,Y 480.891,Z 614.553,A -85,B 0,C 180,E1 21548.247,E2 21548.247} C_VEL
LIN {X 0,Y 485.55,Z 627.341,A -85,B 0,C 180,E1 21546.521,E2 21546.521} C_VEL
LIN {X 0,Y 491.828,Z 645.694,A -85,B 0,C 180,E1 21544.312,E2 21544.312} C_VEL
LIN {X 0,Y 489.321,Z 690.358,A -85,B 0,C 180,E1 21540.492,E2 21540.492} C_VEL
LIN {X 0,Y 488.524,Z 708.782,A -85,B 0,C 180,E1 21538.972,E2 21538.972} C_VEL
LIN {X 0,Y 491.269,Z 729.15,A -85,B 0,C 180,E1 21538.494,E2 21538.494} C_VEL
LIN {X 0,Y 489.135,Z 925.335,A -85,B 0,C 180,E1 21535.526,E2 21535.526} C_VEL
LIN {X 0,Y 488.494,Z 944.832,A -85,B 0,C 180,E1 21535.019,E2 21535.019} C_VEL
LIN {X 0,Y 487.696,Z 963.773,A -85,B 0,C 180,E1 21534.303,E2 21534.303} C_VEL
LIN {X 0,Y 486.78,Z 981.527,A -85,B 0,C 180,E1 21533.419,E2 21533.419} C_VEL
LIN {X 0,Y 485.756,Z 999.043,A -85,B 0,C 180,E1 21532.319,E2 21532.319} C_VEL
LIN {X 0,Y 484.703,Z 1015.705,A -85,B 0,C 180,E1 21531.034,E2 21531.034} C_VEL
LIN {X 0,Y 483.682,Z 1031.465,A -85,B 0,C 180,E1 21529.565,E2 21529.565} C_VEL
LIN {X 0,Y 482.709,Z 1046.241,A -85,B 0,C 180,E1 21527.914,E2 21527.914} C_VEL
LIN {X 0,Y 481.857,Z 1059.726,A -85,B 0,C 180,E1 21526.11,E2 21526.11} C_VEL
LIN {X 0,Y 481.243,Z 1070.006,A -85,B 0,C 180,E1 21524.437,E2 21524.437} C_VEL
LIN {X 0,Y 480.667,Z 1080.3,A -85,B 0,C 180,E1 21522.372,E2 21522.372} C_VEL
LIN {X 0,Y 480.274,Z 1089.028,A -85,B 0,C 180,E1 21520.192,E2 21520.192} C_VEL
LIN {X 0,Y 480.06,Z 1095.822,A -85,B 0,C 180,E1 21518.021,E2 21518.021} C_VEL
LIN {X 0,Y 479.951,Z 1101.086,A -85,B 0,C 180,E1 21515.739,E2 21515.739} C_VEL
LIN {X 0,Y 479.913,Z 1104.538,A -85,B 0,C 180,E1 21513.464,E2 21513.464} C_VEL
LIN {X 0,Y 479.906,Z 1106.266,A -85,B 0,C 180,E1 21511.194,E2 21511.194} C_VEL
LIN {X 0,Y 479.907,Z 1106.303,A -85,B 0,C 180,E1 21508.925,E2 21508.925} C_VEL
LIN {X 0,Y 479.914,Z 1104.656,A -85,B 0,C 180,E1 21506.655,E2 21506.655} C_VEL
LIN {X 0,Y 479.946,Z 1101.292,A -85,B 0,C 180,E1 21504.381,E2 21504.381} C_VEL
LIN {X 0,Y 480.048,Z 1096.123,A -85,B 0,C 180,E1 21502.098,E2 21502.098} C_VEL
LIN {X 0,Y 480.26,Z 1089.43,A -85,B 0,C 180,E1 21499.928,E2 21499.928} C_VEL
LIN {X 0,Y 480.613,Z 1081.336,A -85,B 0,C 180,E1 21497.87,E2 21497.87} C_VEL
LIN {X 0,Y 481.159,Z 1071.296,A -85,B 0,C 180,E1 21495.806,E2 21495.806} C_VEL
LIN {X 0,Y 481.769,Z 1061.112,A -85,B 0,C 180,E1 21494.1,E2 21494.1} C_VEL
LIN {X 0,Y 482.604,Z 1047.719,A -85,B 0,C 180,E1 21492.268,E2 21492.268} C_VEL
LIN {X 0,Y 483.542,Z 1033.539,A -85,B 0,C 180,E1 21490.646,E2 21490.646} C_VEL
LIN {X 0,Y 484.565,Z 1017.967,A -85,B 0,C 180,E1 21489.155,E2 21489.155} C_VEL
LIN {X 0,Y 485.608,Z 1001.734,A -85,B 0,C 180,E1 21487.864,E2 21487.864} C_VEL
LIN {X 0,Y 486.661,Z 984.135,A -85,B 0,C 180,E1 21486.721,E2 21486.721} C_VEL
LIN {X 0,Y 487.607,Z 966.068,A -85,B 0,C 180,E1 21485.788,E2 21485.788} C_VEL
LIN {X 0,Y 488.448,Z 946.92,A -85,B 0,C 180,E1 21485.038,E2 21485.038} C_VEL
LIN {X 0,Y 489.106,Z 927.779,A -85,B 0,C 180,E1 21484.516,E2 21484.516} C_VEL
LIN {X 0,Y 489.552,Z 896.722,A -85,B 0,C 180,E1 21484.007,E2 21484.007} C_VEL
LIN {X 0,Y 491.161,Z 726.445,A -85,B 0,C 180,E1 21481.438,E2 21481.438} C_VEL
LIN {X 0,Y 488.581,Z 708.46,A -85,B 0,C 180,E1 21480.986,E2 21480.986} C_VEL
LIN {X 0,Y 490.529,Z 668.695,A -85,B 0,C 180,E1 21477.652,E2 21477.652} C_VEL
LIN {X 0,Y 491.811,Z 645.304,A -85,B 0,C 180,E1 21475.629,E2 21475.629} C_VEL
LIN {X 0,Y 482.999,Z 620.394,A -85,B 0,C 180,E1 21472.648,E2 21472.648} C_VEL
LIN {X 0,Y 480.898,Z 614.538,A -85,B 0,C 180,E1 21471.865,E2 21471.865} C_VEL
LIN {X 0,Y 480.886,Z 614.332,A -85,B 0,C 180,E1 21468.45,E2 21468.45} C_VEL
LIN {X 0,Y 480.888,Z 614.336,A -85,B 0,C 180,E1 21464.817,E2 21464.817} C_VEL
LIN {X 0,Y 480.881,Z 614.331,A -85,B 0,C 180,E1 21461.176,E2 21461.176} C_VEL
LIN {X 0,Y 480.889,Z 614.331,A -85,B 0,C 180,E1 21457.532,E2 21457.532} C_VEL
LIN {X 0,Y 480.875,Z 614.333,A -85,B 0,C 180,E1 21453.94,E2 21453.94} C_VEL
LIN {X 0,Y 480.882,Z 614.337,A -85,B 0,C 180,E1 21450.348,E2 21450.348} C_VEL
LIN {X 0,Y 480.891,Z 614.333,A -85,B 0,C 180,E1 21446.819,E2 21446.819} C_VEL
LIN {X 0,Y 480.879,Z 614.332,A -85,B 0,C 180,E1 21443.216,E2 21443.216} C_VEL
LIN {X 0,Y 480.857,Z 614.336,A -85,B 0,C 180,E1 21439.619,E2 21439.619} C_VEL
LIN {X 0,Y 480.878,Z 614.338,A -85,B 0,C 180,E1 21436.054,E2 21436.054} C_VEL
LIN {X 0,Y 480.892,Z 614.335,A -85,B 0,C 180,E1 21432.488,E2 21432.488} C_VEL
LIN {X 0,Y 480.845,Z 614.34,A -85,B 0,C 180,E1 21428.972,E2 21428.972} C_VEL
LIN {X 0,Y 480.934,Z 614.67,A -85,B 0,C 180,E1 21428.383,E2 21428.383} C_VEL
LIN {X 0,Y 485.412,Z 631.385,A -85,B 0,C 180,E1 21426.267,E2 21426.267} C_VEL
LIN {X 0,Y 485.991,Z 635.503,A -85,B 0,C 180,E1 21425.786,E2 21425.786} C_VEL
LIN {X 0,Y 485.901,Z 662.457,A -85,B 0,C 180,E1 21422.772,E2 21422.772} C_VEL
LIN {X 0,Y 485.62,Z 688.764,A -85,B 0,C 180,E1 21419.764,E2 21419.764} C_VEL
LIN {X 0,Y 485.42,Z 706.062,A -85,B 0,C 180,E1 21417.775,E2 21417.775} C_VEL
LIN {X 0,Y 485.97,Z 710.504,A -85,B 0,C 180,E1 21417.669,E2 21417.669} C_VEL
LIN {X 0,Y 484.581,Z 845.114,A -85,B 0,C 180,E1 21415.488,E2 21415.488} C_VEL
LIN {X 0,Y 484.442,Z 860.851,A -85,B 0,C 180,E1 21415.019,E2 21415.019} C_VEL
LIN {X 0,Y 484.127,Z 876.815,A -85,B 0,C 180,E1 21414.31,E2 21414.31} C_VEL
LIN {X 0,Y 483.722,Z 890.712,A -85,B 0,C 180,E1 21413.472,E2 21413.472} C_VEL
LIN {X 0,Y 483.183,Z 905.268,A -85,B 0,C 180,E1 21412.33,E2 21412.33} C_VEL
LIN {X 0,Y 482.671,Z 917.05,A -85,B 0,C 180,E1 21411.159,E2 21411.159} C_VEL
LIN {X 0,Y 482.117,Z 928.606,A -85,B 0,C 180,E1 21409.726,E2 21409.726} C_VEL
LIN {X 0,Y 481.655,Z 938.083,A -85,B 0,C 180,E1 21408.262,E2 21408.262} C_VEL
LIN {X 0,Y 481.229,Z 946.991,A -85,B 0,C 180,E1 21406.503,E2 21406.503} C_VEL
LIN {X 0,Y 480.931,Z 953.867,A -85,B 0,C 180,E1 21404.724,E2 21404.724} C_VEL
LIN {X 0,Y 480.709,Z 959.161,A -85,B 0,C 180,E1 21402.821,E2 21402.821} C_VEL
LIN {X 0,Y 480.578,Z 962.563,A -85,B 0,C 180,E1 21400.935,E2 21400.935} C_VEL
LIN {X 0,Y 480.511,Z 964.301,A -85,B 0,C 180,E1 21398.901,E2 21398.901} C_VEL
LIN {X 0,Y 480.497,Z 964.17,A -85,B 0,C 180,E1 21396.97,E2 21396.97} C_VEL
LIN {X 0,Y 480.527,Z 962.269,A -85,B 0,C 180,E1 21395.014,E2 21395.014} C_VEL
LIN {X 0,Y 480.62,Z 958.799,A -85,B 0,C 180,E1 21393.164,E2 21393.164} C_VEL
LIN {X 0,Y 480.793,Z 953.452,A -85,B 0,C 180,E1 21391.289,E2 21391.289} C_VEL
LIN {X 0,Y 481.06,Z 946.6,A -85,B 0,C 180,E1 21389.526,E2 21389.526} C_VEL
LIN {X 0,Y 481.447,Z 937.477,A -85,B 0,C 180,E1 21387.742,E2 21387.742} C_VEL
LIN {X 0,Y 481.906,Z 927.579,A -85,B 0,C 180,E1 21386.217,E2 21386.217} C_VEL
LIN {X 0,Y 482.463,Z 915.533,A -85,B 0,C 180,E1 21384.739,E2 21384.739} C_VEL
LIN {X 0,Y 482.986,Z 903.419,A -85,B 0,C 180,E1 21383.549,E2 21383.549} C_VEL
LIN {X 0,Y 483.547,Z 888.75,A -85,B 0,C 180,E1 21382.411,E2 21382.411} C_VEL
LIN {X 0,Y 483.81,Z 880.709,A -85,B 0,C 180,E1 21381.901,E2 21381.901} C_VEL
LIN {X 0,Y 483.136,Z 873.78,A -85,B 0,C 180,E1 21381.488,E2 21381.488} C_VEL
LIN {X 0,Y 478.546,Z 859.234,A -85,B 0,C 180,E1 21380.655,E2 21380.655} C_VEL
LIN {X 0,Y 477.046,Z 852.049,A -85,B 0,C 180,E1 21380.351,E2 21380.351} C_VEL
LIN {X 0,Y 476.859,Z 848.838,A -85,B 0,C 180,E1 21380.252,E2 21380.252} C_VEL
LIN {X 0,Y 476.956,Z 831.065,A -85,B 0,C 180,E1 21379.886,E2 21379.886} C_VEL
LIN {X 0,Y 478.091,Z 708.553,A -85,B 0,C 180,E1 21377.923,E2 21377.923} C_VEL
LIN {X 0,Y 476.933,Z 702.3,A -85,B 0,C 180,E1 21377.735,E2 21377.735} C_VEL
LIN {X 0,Y 477.593,Z 672.903,A -85,B 0,C 180,E1 21374.199,E2 21374.199} C_VEL
LIN {X 0,Y 478.181,Z 642.855,A -85,B 0,C 180,E1 21370.622,E2 21370.622} C_VEL
LIN {X 0,Y 478.154,Z 635.848,A -85,B 0,C 180,E1 21369.783,E2 21369.783} C_VEL
LIN {X 0,Y 473.586,Z 617.962,A -85,B 0,C 180,E1 21367.372,E2 21367.372} C_VEL
LIN {X 0,Y 472.901,Z 615.423,A -85,B 0,C 180,E1 21366.945,E2 21366.945} C_VEL
LIN {X 0,Y 472.943,Z 615.313,A -85,B 0,C 180,E1 21363.49,E2 21363.49} C_VEL
LIN {X 0,Y 472.906,Z 615.326,A -85,B 0,C 180,E1 21360.072,E2 21360.072} C_VEL
LIN {X 0,Y 472.897,Z 615.323,A -85,B 0,C 180,E1 21356.496,E2 21356.496} C_VEL
LIN {X 0,Y 472.948,Z 615.314,A -85,B 0,C 180,E1 21353.024,E2 21353.024} C_VEL
LIN {X 0,Y 472.925,Z 615.305,A -85,B 0,C 180,E1 21349.449,E2 21349.449} C_VEL
LIN {X 0,Y 472.9,Z 615.308,A -85,B 0,C 180,E1 21345.954,E2 21345.954} C_VEL
LIN {X 0,Y 472.981,Z 615.663,A -85,B 0,C 180,E1 21345.289,E2 21345.289} C_VEL
LIN {X 0,Y 477.973,Z 633.612,A -85,B 0,C 180,E1 21342.32,E2 21342.32} C_VEL
LIN {X 0,Y 479.625,Z 640.807,A -85,B 0,C 180,E1 21341.179,E2 21341.179} C_VEL
LIN {X 0,Y 478.075,Z 668.165,A -85,B 0,C 180,E1 21337.451,E2 21337.451} C_VEL
LIN {X 0,Y 476.796,Z 693.879,A -85,B 0,C 180,E1 21334.029,E2 21334.029} C_VEL
LIN {X 0,Y 480.301,Z 711.656,A -85,B 0,C 180,E1 21333.532,E2 21333.532} C_VEL
LIN {X 0,Y 478.849,Z 839.699,A -85,B 0,C 180,E1 21331.518,E2 21331.518} C_VEL
LIN {X 0,Y 478.488,Z 856.677,A -85,B 0,C 180,E1 21331.014,E2 21331.014} C_VEL
LIN {X 0,Y 477.992,Z 871.652,A -85,B 0,C 180,E1 21330.36,E2 21330.36} C_VEL
LIN {X 0,Y 477.295,Z 886.79,A -85,B 0,C 180,E1 21329.46,E2 21329.46} C_VEL
LIN {X 0,Y 476.481,Z 901.618,A -85,B 0,C 180,E1 21328.317,E2 21328.317} C_VEL
LIN {X 0,Y 475.693,Z 914.524,A -85,B 0,C 180,E1 21327.048,E2 21327.048} C_VEL
LIN {X 0,Y 474.878,Z 926.856,A -85,B 0,C 180,E1 21325.532,E2 21325.532} C_VEL
LIN {X 0,Y 474.179,Z 937.139,A -85,B 0,C 180,E1 21323.948,E2 21323.948} C_VEL
LIN {X 0,Y 473.564,Z 946.517,A -85,B 0,C 180,E1 21322.112,E2 21322.112} C_VEL
LIN {X 0,Y 473.145,Z 953.76,A -85,B 0,C 180,E1 21320.267,E2 21320.267} C_VEL
LIN {X 0,Y 472.85,Z 959.529,A -85,B 0,C 180,E1 21318.248,E2 21318.248} C_VEL
LIN {X 0,Y 472.684,Z 963.281,A -85,B 0,C 180,E1 21316.296,E2 21316.296} C_VEL
LIN {X 0,Y 472.6,Z 965.313,A -85,B 0,C 180,E1 21314.287,E2 21314.287} C_VEL
LIN {X 0,Y 472.603,Z 965.658,A -85,B 0,C 180,E1 21312.184,E2 21312.184} C_VEL
LIN {X 0,Y 472.676,Z 964.244,A -85,B 0,C 180,E1 21310.218,E2 21310.218} C_VEL
LIN {X 0,Y 472.849,Z 960.956,A -85,B 0,C 180,E1 21308.151,E2 21308.151} C_VEL
LIN {X 0,Y 473.129,Z 956.016,A -85,B 0,C 180,E1 21306.194,E2 21306.194} C_VEL
LIN {X 0,Y 473.566,Z 948.984,A -85,B 0,C 180,E1 21304.219,E2 21304.219} C_VEL
LIN {X 0,Y 474.131,Z 940.957,A -85,B 0,C 180,E1 21302.495,E2 21302.495} C_VEL
LIN {X 0,Y 474.849,Z 931.031,A -85,B 0,C 180,E1 21300.827,E2 21300.827} C_VEL
LIN {X 0,Y 475.686,Z 919.564,A -85,B 0,C 180,E1 21299.282,E2 21299.282} C_VEL
LIN {X 0,Y 476.525,Z 907.008,A -85,B 0,C 180,E1 21297.937,E2 21297.937} C_VEL
LIN {X 0,Y 477.401,Z 892.719,A -85,B 0,C 180,E1 21296.721,E2 21296.721} C_VEL
LIN {X 0,Y 478.147,Z 878.388,A -85,B 0,C 180,E1 21295.771,E2 21295.771} C_VEL
LIN {X 0,Y 478.786,Z 862.656,A -85,B 0,C 180,E1 21294.987,E2 21294.987} C_VEL
LIN {X 0,Y 479.227,Z 846.358,A -85,B 0,C 180,E1 21294.416,E2 21294.416} C_VEL
LIN {X 0,Y 479.465,Z 827.655,A -85,B 0,C 180,E1 21294.034,E2 21294.034} C_VEL
LIN {X 0,Y 480.813,Z 710.287,A -85,B 0,C 180,E1 21292.17,E2 21292.17} C_VEL
LIN {X 0,Y 477.373,Z 694.562,A -85,B 0,C 180,E1 21291.686,E2 21291.686} C_VEL
LIN {X 0,Y 477.607,Z 688.117,A -85,B 0,C 180,E1 21290.863,E2 21290.863} C_VEL
LIN {X 0,Y 479.325,Z 659.935,A -85,B 0,C 180,E1 21286.991,E2 21286.991} C_VEL
LIN {X 0,Y 480.535,Z 641.839,A -85,B 0,C 180,E1 21284.465,E2 21284.465} C_VEL
LIN {X 0,Y 476.394,Z 626.594,A -85,B 0,C 180,E1 21281.835,E2 21281.835} C_VEL
LIN {X 0,Y 472.971,Z 615.44,A -85,B 0,C 180,E1 21279.754,E2 21279.754} C_VEL
LIN {X 0,Y 472.941,Z 615.32,A -85,B 0,C 180,E1 21276.138,E2 21276.138} C_VEL
LIN {X 0,Y 472.949,Z 615.325,A -85,B 0,C 180,E1 21272.479,E2 21272.479} C_VEL
LIN {X 0,Y 472.943,Z 615.318,A -85,B 0,C 180,E1 21268.818,E2 21268.818} C_VEL
LIN {X 0,Y 472.949,Z 615.315,A -85,B 0,C 180,E1 21265.147,E2 21265.147} C_VEL
LIN {X 0,Y 472.939,Z 615.32,A -85,B 0,C 180,E1 21261.531,E2 21261.531} C_VEL
LIN {X 0,Y 472.948,Z 615.316,A -85,B 0,C 180,E1 21257.851,E2 21257.851} C_VEL
LIN {X 0,Y 472.943,Z 615.312,A -85,B 0,C 180,E1 21254.196,E2 21254.196} C_VEL
LIN {X 0,Y 472.945,Z 615.312,A -85,B 0,C 180,E1 21250.562,E2 21250.562} C_VEL
LIN {X 0,Y 472.934,Z 615.319,A -85,B 0,C 180,E1 21246.922,E2 21246.922} C_VEL
LIN {X 0,Y 472.947,Z 615.325,A -85,B 0,C 180,E1 21243.273,E2 21243.273} C_VEL
LIN {X 0,Y 472.946,Z 615.313,A -85,B 0,C 180,E1 21239.558,E2 21239.558} C_VEL
LIN {X 0,Y 472.945,Z 615.307,A -85,B 0,C 180,E1 21235.878,E2 21235.878} C_VEL
LIN {X 0,Y 472.931,Z 615.316,A -85,B 0,C 180,E1 21232.224,E2 21232.224} C_VEL
LIN {X 0,Y 472.944,Z 615.325,A -85,B 0,C 180,E1 21228.538,E2 21228.538} C_VEL
LIN {X 0,Y 472.947,Z 615.313,A -85,B 0,C 180,E1 21224.928,E2 21224.928} C_VEL
LIN {X 0,Y 472.944,Z 615.307,A -85,B 0,C 180,E1 21221.256,E2 21221.256} C_VEL
LIN {X 0,Y 472.927,Z 615.315,A -85,B 0,C 180,E1 21217.632,E2 21217.632} C_VEL
LIN {X 0,Y 472.944,Z 615.32,A -85,B 0,C 180,E1 21213.961,E2 21213.961} C_VEL
LIN {X 0,Y 472.952,Z 615.323,A -85,B 0,C 180,E1 21210.329,E2 21210.329} C_VEL
LIN {X 0,Y 472.944,Z 615.321,A -85,B 0,C 180,E1 21206.656,E2 21206.656} C_VEL
LIN {X 0,Y 472.926,Z 615.322,A -85,B 0,C 180,E1 21203.05,E2 21203.05} C_VEL
LIN {X 0,Y 472.954,Z 615.319,A -85,B 0,C 180,E1 21199.532,E2 21199.532} C_VEL
LIN {X 0,Y 472.951,Z 615.316,A -85,B 0,C 180,E1 21195.93,E2 21195.93} C_VEL
LIN {X 0,Y 472.924,Z 615.325,A -85,B 0,C 180,E1 21192.41,E2 21192.41} C_VEL
LIN {X 0,Y 472.975,Z 615.572,A -85,B 0,C 180,E1 21188.867,E2 21188.867} C_VEL
LIN {X 0,Y 476.098,Z 624.03,A -85,B 0,C 180,E1 21187.652,E2 21187.652} C_VEL
LIN {X 0,Y 482.795,Z 643.152,A -85,B 0,C 180,E1 21185.214,E2 21185.214} C_VEL
LIN {X 0,Y 484.564,Z 648.535,A -85,B 0,C 180,E1 21184.572,E2 21184.572} C_VEL
LIN {X 0,Y 481.879,Z 692.178,A -85,B 0,C 180,E1 21180.768,E2 21180.768} C_VEL
LIN {X 0,Y 481.092,Z 708.787,A -85,B 0,C 180,E1 21179.372,E2 21179.372} C_VEL
LIN {X 0,Y 483.954,Z 730.212,A -85,B 0,C 180,E1 21178.864,E2 21178.864} C_VEL
LIN {X 0,Y 481.673,Z 924.499,A -85,B 0,C 180,E1 21175.881,E2 21175.881} C_VEL
LIN {X 0,Y 480.995,Z 943.998,A -85,B 0,C 180,E1 21175.367,E2 21175.367} C_VEL
LIN {X 0,Y 480.162,Z 962.424,A -85,B 0,C 180,E1 21174.665,E2 21174.665} C_VEL
LIN {X 0,Y 479.153,Z 980.585,A -85,B 0,C 180,E1 21173.749,E2 21173.749} C_VEL
LIN {X 0,Y 478.066,Z 998.096,A -85,B 0,C 180,E1 21172.633,E2 21172.633} C_VEL
LIN {X 0,Y 476.958,Z 1014.588,A -85,B 0,C 180,E1 21171.343,E2 21171.343} C_VEL
LIN {X 0,Y 475.858,Z 1030.494,A -85,B 0,C 180,E1 21169.836,E2 21169.836} C_VEL
LIN {X 0,Y 474.831,Z 1045.251,A -85,B 0,C 180,E1 21168.158,E2 21168.158} C_VEL
LIN {X 0,Y 473.983,Z 1058.097,A -85,B 0,C 180,E1 21166.419,E2 21166.419} C_VEL
LIN {X 0,Y 473.236,Z 1070.308,A -85,B 0,C 180,E1 21164.436,E2 21164.436} C_VEL
LIN {X 0,Y 472.691,Z 1080.394,A -85,B 0,C 180,E1 21162.46,E2 21162.46} C_VEL
LIN {X 0,Y 472.332,Z 1088.538,A -85,B 0,C 180,E1 21160.489,E2 21160.489} C_VEL
LIN {X 0,Y 472.096,Z 1095.127,A -85,B 0,C 180,E1 21158.403,E2 21158.403} C_VEL
LIN {X 0,Y 471.967,Z 1100.341,A -85,B 0,C 180,E1 21156.202,E2 21156.202} C_VEL
LIN {X 0,Y 471.92,Z 1103.911,A -85,B 0,C 180,E1 21154.009,E2 21154.009} C_VEL
LIN {X 0,Y 471.911,Z 1105.996,A -85,B 0,C 180,E1 21151.699,E2 21151.699} C_VEL
LIN {X 0,Y 471.909,Z 1106.393,A -85,B 0,C 180,E1 21149.393,E2 21149.393} C_VEL
LIN {X 0,Y 471.909,Z 1105.11,A -85,B 0,C 180,E1 21147.085,E2 21147.085} C_VEL
LIN {X 0,Y 471.936,Z 1102.027,A -85,B 0,C 180,E1 21144.719,E2 21144.719} C_VEL
LIN {X 0,Y 472.029,Z 1097.319,A -85,B 0,C 180,E1 21142.446,E2 21142.446} C_VEL
LIN {X 0,Y 472.25,Z 1090.632,A -85,B 0,C 180,E1 21140.125,E2 21140.125} C_VEL
LIN {X 0,Y 472.56,Z 1083.116,A -85,B 0,C 180,E1 21138.156,E2 21138.156} C_VEL
LIN {X 0,Y 473.077,Z 1073.008,A -85,B 0,C 180,E1 21136.058,E2 21136.058} C_VEL
LIN {X 0,Y 473.771,Z 1061.386,A -85,B 0,C 180,E1 21134.076,E2 21134.076} C_VEL
LIN {X 0,Y 474.625,Z 1048.241,A -85,B 0,C 180,E1 21132.212,E2 21132.212} C_VEL
LIN {X 0,Y 475.655,Z 1033.532,A -85,B 0,C 180,E1 21130.474,E2 21130.474} C_VEL
LIN {X 0,Y 476.731,Z 1018.136,A -85,B 0,C 180,E1 21128.956,E2 21128.956} C_VEL
LIN {X 0,Y 477.912,Z 1000.891,A -85,B 0,C 180,E1 21127.553,E2 21127.553} C_VEL
LIN {X 0,Y 479.055,Z 983.02,A -85,B 0,C 180,E1 21126.376,E2 21126.376} C_VEL
LIN {X 0,Y 480.092,Z 964.61,A -85,B 0,C 180,E1 21125.417,E2 21125.417} C_VEL
LIN {X 0,Y 480.969,Z 945.695,A -85,B 0,C 180,E1 21124.672,E2 21124.672} C_VEL
LIN {X 0,Y 481.667,Z 926.647,A -85,B 0,C 180,E1 21124.151,E2 21124.151} C_VEL
LIN {X 0,Y 482.157,Z 893.456,A -85,B 0,C 180,E1 21123.606,E2 21123.606} C_VEL
LIN {X 0,Y 483.876,Z 727.599,A -85,B 0,C 180,E1 21121.066,E2 21121.066} C_VEL
LIN {X 0,Y 481.15,Z 708.641,A -85,B 0,C 180,E1 21120.597,E2 21120.597} C_VEL
LIN {X 0,Y 483.351,Z 668.032,A -85,B 0,C 180,E1 21117.124,E2 21117.124} C_VEL
LIN {X 0,Y 484.591,Z 648.406,A -85,B 0,C 180,E1 21115.412,E2 21115.412} C_VEL
LIN {X 0,Y 476.224,Z 624.58,A -85,B 0,C 180,E1 21112.526,E2 21112.526} C_VEL
LIN {X 0,Y 472.968,Z 615.532,A -85,B 0,C 180,E1 21111.318,E2 21111.318} C_VEL
LIN {X 0,Y 472.937,Z 615.32,A -85,B 0,C 180,E1 21107.727,E2 21107.727} C_VEL
LIN {X 0,Y 472.949,Z 615.317,A -85,B 0,C 180,E1 21104.07,E2 21104.07} C_VEL
LIN {X 0,Y 472.943,Z 615.325,A -85,B 0,C 180,E1 21100.44,E2 21100.44} C_VEL
LIN {X 0,Y 472.949,Z 615.325,A -85,B 0,C 180,E1 21096.899,E2 21096.899} C_VEL
LIN {X 0,Y 472.948,Z 615.322,A -85,B 0,C 180,E1 21093.199,E2 21093.199} C_VEL
LIN {X 0,Y 472.937,Z 615.32,A -85,B 0,C 180,E1 21089.65,E2 21089.65} C_VEL
LIN {X 0,Y 472.929,Z 615.326,A -85,B 0,C 180,E1 21085.953,E2 21085.953} C_VEL
LIN {X 0,Y 472.954,Z 615.325,A -85,B 0,C 180,E1 21082.367,E2 21082.367} C_VEL
LIN {X 0,Y 472.954,Z 615.322,A -85,B 0,C 180,E1 21078.718,E2 21078.718} C_VEL
LIN {X 0,Y 472.914,Z 615.327,A -85,B 0,C 180,E1 21075.199,E2 21075.199} C_VEL
LIN {X 0,Y 472.913,Z 615.328,A -85,B 0,C 180,E1 21071.587,E2 21071.587} C_VEL
LIN {X 0,Y 472.944,Z 615.558,A -85,B 0,C 180,E1 21068.847,E2 21068.847} C_VEL
LIN {X 0,Y 477.677,Z 632.401,A -85,B 0,C 180,E1 21066.671,E2 21066.671} C_VEL
LIN {X 0,Y 478.585,Z 637.727,A -85,B 0,C 180,E1 21066.03,E2 21066.03} C_VEL
LIN {X 0,Y 478.461,Z 665.841,A -85,B 0,C 180,E1 21062.875,E2 21062.875} C_VEL
LIN {X 0,Y 478.152,Z 691.96,A -85,B 0,C 180,E1 21059.88,E2 21059.88} C_VEL
LIN {X 0,Y 477.988,Z 707.501,A -85,B 0,C 180,E1 21058.097,E2 21058.097} C_VEL
LIN {X 0,Y 478.494,Z 711.761,A -85,B 0,C 180,E1 21057.994,E2 21057.994} C_VEL
LIN {X 0,Y 476.967,Z 846.499,A -85,B 0,C 180,E1 21055.755,E2 21055.755} C_VEL
LIN {X 0,Y 476.824,Z 862.401,A -85,B 0,C 180,E1 21055.271,E2 21055.271} C_VEL
LIN {X 0,Y 476.509,Z 877.715,A -85,B 0,C 180,E1 21054.582,E2 21054.582} C_VEL
LIN {X 0,Y 476.088,Z 891.737,A -85,B 0,C 180,E1 21053.73,E2 21053.73} C_VEL
LIN {X 0,Y 475.541,Z 905.658,A -85,B 0,C 180,E1 21052.631,E2 21052.631} C_VEL
LIN {X 0,Y 474.982,Z 917.984,A -85,B 0,C 180,E1 21051.404,E2 21051.404} C_VEL
LIN {X 0,Y 474.373,Z 929.764,A -85,B 0,C 180,E1 21049.924,E2 21049.924} C_VEL
LIN {X 0,Y 473.872,Z 939.266,A -85,B 0,C 180,E1 21048.437,E2 21048.437} C_VEL
LIN {X 0,Y 473.414,Z 948.002,A -85,B 0,C 180,E1 21046.69,E2 21046.69} C_VEL
LIN {X 0,Y 473.096,Z 954.793,A -85,B 0,C 180,E1 21044.932,E2 21044.932} C_VEL
LIN {X 0,Y 472.84,Z 960.089,A -85,B 0,C 180,E1 21043.033,E2 21043.033} C_VEL
LIN {X 0,Y 472.693,Z 963.63,A -85,B 0,C 180,E1 21041.117,E2 21041.117} C_VEL
LIN {X 0,Y 472.613,Z 965.397,A -85,B 0,C 180,E1 21039.18,E2 21039.18} C_VEL
LIN {X 0,Y 472.587,Z 965.501,A -85,B 0,C 180,E1 21037.221,E2 21037.221} C_VEL
LIN {X 0,Y 472.613,Z 963.805,A -85,B 0,C 180,E1 21035.235,E2 21035.235} C_VEL
LIN {X 0,Y 472.717,Z 960.218,A -85,B 0,C 180,E1 21033.201,E2 21033.201} C_VEL
LIN {X 0,Y 472.898,Z 955.015,A -85,B 0,C 180,E1 21031.317,E2 21031.317} C_VEL
LIN {X 0,Y 473.181,Z 948.274,A -85,B 0,C 180,E1 21029.527,E2 21029.527} C_VEL
LIN {X 0,Y 473.552,Z 940.058,A -85,B 0,C 180,E1 21027.852,E2 21027.852} C_VEL
LIN {X 0,Y 474.074,Z 929.562,A -85,B 0,C 180,E1 21026.165,E2 21026.165} C_VEL
LIN {X 0,Y 474.62,Z 918.394,A -85,B 0,C 180,E1 21024.744,E2 21024.744} C_VEL
LIN {X 0,Y 475.209,Z 905.831,A -85,B 0,C 180,E1 21023.455,E2 21023.455} C_VEL
LIN {X 0,Y 475.766,Z 892.255,A -85,B 0,C 180,E1 21022.353,E2 21022.353} C_VEL
LIN {X 0,Y 476.287,Z 876.917,A -85,B 0,C 180,E1 21021.385,E2 21021.385} C_VEL
LIN {X 0,Y 476.671,Z 861.166,A -85,B 0,C 180,E1 21020.66,E2 21020.66} C_VEL
LIN {X 0,Y 476.859,Z 848.838,A -85,B 0,C 180,E1 21020.252,E2 21020.252} C_VEL
LIN {X 0,Y 475.988,Z 841.335,A -85,B 0,C 180,E1 21020.033,E2 21020.033} C_VEL
LIN {X 0,Y 470.117,Z 821.476,A -85,B 0,C 180,E1 21019.466,E2 21019.466} C_VEL
LIN {X 0,Y 469.47,Z 814.945,A -85,B 0,C 180,E1 21019.337,E2 21019.337} C_VEL
LIN {X 0,Y 470.575,Z 709.743,A -85,B 0,C 180,E1 21017.609,E2 21017.609} C_VEL
LIN {X 0,Y 469.376,Z 703.323,A -85,B 0,C 180,E1 21017.421,E2 21017.421} C_VEL
LIN {X 0,Y 470.022,Z 674.099,A -85,B 0,C 180,E1 21013.907,E2 21013.907} C_VEL
LIN {X 0,Y 470.654,Z 644.748,A -85,B 0,C 180,E1 21010.387,E2 21010.387} C_VEL
LIN {X 0,Y 470.466,Z 637.514,A -85,B 0,C 180,E1 21009.514,E2 21009.514} C_VEL
LIN {X 0,Y 465.58,Z 618.782,A -85,B 0,C 180,E1 21006.965,E2 21006.965} C_VEL
LIN {X 0,Y 464.965,Z 616.421,A -85,B 0,C 180,E1 21006.56,E2 21006.56} C_VEL
LIN {X 0,Y 464.962,Z 616.307,A -85,B 0,C 180,E1 21002.96,E2 21002.96} C_VEL
LIN {X 0,Y 465.02,Z 616.311,A -85,B 0,C 180,E1 20999.447,E2 20999.447} C_VEL
LIN {X 0,Y 464.969,Z 616.301,A -85,B 0,C 180,E1 20995.883,E2 20995.883} C_VEL
LIN {X 0,Y 464.959,Z 616.317,A -85,B 0,C 180,E1 20992.24,E2 20992.24} C_VEL
LIN {X 0,Y 464.993,Z 616.3,A -85,B 0,C 180,E1 20988.687,E2 20988.687} C_VEL
LIN {X 0,Y 464.999,Z 616.555,A -85,B 0,C 180,E1 20985.8,E2 20985.8} C_VEL
LIN {X 0,Y 470.297,Z 635.436,A -85,B 0,C 180,E1 20982.618,E2 20982.618} C_VEL
LIN {X 0,Y 472.113,Z 643.244,A -85,B 0,C 180,E1 20981.36,E2 20981.36} C_VEL
LIN {X 0,Y 470.525,Z 669.885,A -85,B 0,C 180,E1 20977.694,E2 20977.694} C_VEL
LIN {X 0,Y 469.238,Z 694.14,A -85,B 0,C 180,E1 20974.43,E2 20974.43} C_VEL
LIN {X 0,Y 472.963,Z 712.886,A -85,B 0,C 180,E1 20973.902,E2 20973.902} C_VEL
LIN {X 0,Y 471.416,Z 840.456,A -85,B 0,C 180,E1 20971.865,E2 20971.865} C_VEL
LIN {X 0,Y 471.036,Z 857.477,A -85,B 0,C 180,E1 20971.352,E2 20971.352} C_VEL
LIN {X 0,Y 470.498,Z 872.825,A -85,B 0,C 180,E1 20970.67,E2 20970.67} C_VEL
LIN {X 0,Y 469.759,Z 887.898,A -85,B 0,C 180,E1 20969.756,E2 20969.756} C_VEL
LIN {X 0,Y 468.933,Z 901.991,A -85,B 0,C 180,E1 20968.656,E2 20968.656} C_VEL
LIN {X 0,Y 468.09,Z 915.047,A -85,B 0,C 180,E1 20967.368,E2 20967.368} C_VEL
LIN {X 0,Y 467.208,Z 927.468,A -85,B 0,C 180,E1 20965.828,E2 20965.828} C_VEL
LIN {X 0,Y 466.45,Z 937.864,A -85,B 0,C 180,E1 20964.218,E2 20964.218} C_VEL
LIN {X 0,Y 465.812,Z 946.75,A -85,B 0,C 180,E1 20962.477,E2 20962.477} C_VEL
LIN {X 0,Y 465.334,Z 954.221,A -85,B 0,C 180,E1 20960.602,E2 20960.602} C_VEL
LIN {X 0,Y 465.006,Z 959.911,A -85,B 0,C 180,E1 20958.666,E2 20958.666} C_VEL
LIN {X 0,Y 464.795,Z 964.119,A -85,B 0,C 180,E1 20956.566,E2 20956.566} C_VEL
LIN {X 0,Y 464.697,Z 966.373,A -85,B 0,C 180,E1 20954.526,E2 20954.526} C_VEL
LIN {X 0,Y 464.689,Z 966.876,A -85,B 0,C 180,E1 20952.339,E2 20952.339} C_VEL
LIN {X 0,Y 464.773,Z 965.573,A -85,B 0,C 180,E1 20950.26,E2 20950.26} C_VEL
LIN {X 0,Y 464.96,Z 962.379,A -85,B 0,C 180,E1 20948.16,E2 20948.16} C_VEL
LIN {X 0,Y 465.271,Z 957.586,A -85,B 0,C 180,E1 20946.171,E2 20946.171} C_VEL
LIN {X 0,Y 465.7,Z 951.215,A -85,B 0,C 180,E1 20944.298,E2 20944.298} C_VEL
LIN {X 0,Y 466.345,Z 942.808,A -85,B 0,C 180,E1 20942.412,E2 20942.412} C_VEL
LIN {X 0,Y 467.11,Z 933.201,A -85,B 0,C 180,E1 20940.731,E2 20940.731} C_VEL
LIN {X 0,Y 468.049,Z 921.312,A -85,B 0,C 180,E1 20939.079,E2 20939.079} C_VEL
LIN {X 0,Y 468.938,Z 909.346,A -85,B 0,C 180,E1 20937.747,E2 20937.747} C_VEL
LIN {X 0,Y 469.851,Z 895.632,A -85,B 0,C 180,E1 20936.532,E2 20936.532} C_VEL
LIN {X 0,Y 470.696,Z 880.936,A -85,B 0,C 180,E1 20935.508,E2 20935.508} C_VEL
LIN {X 0,Y 471.365,Z 866.174,A -85,B 0,C 180,E1 20934.729,E2 20934.729} C_VEL
LIN {X 0,Y 471.881,Z 849.207,A -85,B 0,C 180,E1 20934.094,E2 20934.094} C_VEL
LIN {X 0,Y 472.143,Z 832.439,A -85,B 0,C 180,E1 20933.708,E2 20933.708} C_VEL
LIN {X 0,Y 473.616,Z 711.458,A -85,B 0,C 180,E1 20931.752,E2 20931.752} C_VEL
LIN {X 0,Y 469.963,Z 694.976,A -85,B 0,C 180,E1 20931.237,E2 20931.237} C_VEL
